(* IEC 61131-3 sources: elnaProjects/kc6/build_BaseProject_ecl/_ (part 4) *)

  errorCMDTimer(In := _commandErrorTimer, PT :=T#90s);

  continueHoldCommandTimer(IN:=(strKr.onStatus = _statusDualInput.STATUS_ON) OR
  (strKr.onStatus = _statusDualInput.STATUS_OFF), PT:=strKr.continueHoldCommand);

  (* ---- алгоритм  для команды ВКЛючить ---- *)
  IF (strKr.onStatus = _statusDualInput.STATUS_ON) and strKr.lastCmdIsOn  then
  	IF strKr.ISVALIDREF_cmdOn AND strKr.ISVALIDREF_cmdOff then
            IF continueHoldCommandTimer.Q THEN
            strKr.cmdOn := false; END_IF;
            END_IF;
  	 errorCMDTimer(In := false);
  	 _commandErrorTimer := false;
  	 cmd_for_Status := 0;
  	 source_for_Status := 0;
  END_IF;

  (* ---- off ---- *)
  IF (strKr.onStatus = _statusDualInput.STATUS_OFF) and  (NOT strKr.lastCmdIsOn) then
  	IF strKr.ISVALIDREF_cmdOn AND strKr.ISVALIDREF_cmdOff then
            IF continueHoldCommandTimer.Q THEN
            strKr.cmdOff := false; END_IF;
            END_IF;
  	 errorCMDTimer(In := false);
  	 _commandErrorTimer := false;
  	 cmd_for_Status := 0;
  	 source_for_Status := 0;
  END_IF;

  (* ---- ошибка исполнения команды ---- *)
  if errorCMDTimer.Q and (cmd_for_Status <> 0) then
  	command_error_for_Status :=  cmd_for_Status;
  	_commandErrorTimer := false;
  	strKr.CmdOn := false;
  	strKr.CmdOff := false;
  	(*lastCmd := 0;*)
  END_IF;

  (* ---- сброс ошибки команды ---- *)
  strKr.CommandFault := command_error_for_Status <> 0;
  _errorReset(IN := command_error_for_Status <> 0, PT := T#5S);
  IF _errorReset.Q THEN
  	cmd_for_Status := 0;
  	source_for_Status := 0;
  	command_error_for_Status := 0;

  END_IF;

  outputsSets(in := (strKr.ISVALIDREF_cmdOn and strKr.cmdOn ) OR (strKr.ISVALIDREF_cmdOff and strKr.cmdOff), PT := T#2S);
  	IF NOT outputsSets.Q THEN
  		strKr.So := inSo._inversed AND inSo.reliability AND strKr.ISVALIDREF_inSo;
  		strKr.Sz := inSz._inversed AND inSz.reliability AND strKr.ISVALIDREF_inSz;
  	END_IF;

  cmdOn := strKr.cmdOn;
  cmdOff:= strKr.cmdOff;

  (* ---- формирование зашифрованного статуса для АРМа ---- *)
  strKr.status := shl(BYTE_TO_DWORD(source_for_Status), 29)
  		OR shl(BYTE_TO_DWORD(cmd_for_Status), 26)
  		OR shl(BYTE_TO_DWORD(command_error_for_Status), 23)
  		OR shl(bool_to_DWORD(strKr.sdvig), 22)
  		OR shl(bool_to_DWORD(strKr.OpcCommandsDisabled), 21)
                      OR shl(bool_to_DWORD(strKr.Dp), 14)
                      OR shl(BOOL_TO_DWORD(strKr.Sz), 13)
  		OR shl(BOOL_TO_DWORD(strKr.So), 12)
  		OR shl(BOOL_TO_DWORD(strKr.ErrorBlock), 11)
  		OR shl(BOOL_TO_DWORD(strKr.ErrorPowerOff), 10)
  		OR shl(BOOL_TO_DWORD(strKr.Manual), 8)
  		OR shl(BOOL_TO_DWORD(strKr.Auto), 7)
  		OR shl(BOOL_TO_DWORD(strKr.Distance), 6)
  		OR shl(BOOL_TO_DWORD(strKr.Local), 5)
  		OR shl(BOOL_TO_DWORD(strKr.Ns), 4)
                  	OR shl(BOOL_TO_DWORD(strKr.Accident ),3)
  		OR BYTE_TO_DWORD(strKr.onStatus);
END_FUNCTION_BLOCK

FUNCTION_BLOCK fb_KranOpenProtectionDual
  VAR_INPUT
    im : struct_Kran;
    dp_konf : struct_AI;
    parametr : struct_DiscretParametr;
  END_VAR
  VAR_IN_OUT
    StrDIp : struct_DiProtection;
  END_VAR
  VAR
    _sunpackerCommand : fb_sunpackerCommand;
    statusDualInput : TYPE_statusDualInput;
    _statusAi : TYPE_StatusAi;
    _ProtectionTags : TYPE_ProtectionTags;
    dP_Konf_izm : LREAL;
    _signalingTp : TOF;
    timer : TON;
    SignalingTrig : R_TRIG;
    SignalingFTrig : F_TRIG;
    SignalingDi : BOOL;
    _signaling : BOOL;
    source : BYTE;
    cmd : BYTE;
    lastCmd : BYTE;
    source_for_Status : BYTE;
    cmd_for_Status : BYTE;
    command_error_for_Status : BYTE;
    resetCmdTimer : TON;
    resetCmdTimerPriznak : BOOL;
    signalinTimer : TON;
    runOnStart_Trig : R_TRIG;
  END_VAR

  IF parametr.Value = 0 THEN
  	dP_Konf_izm:=0.0;
  	timer (in:=(im.onStatus <> statusDualInput.status_on AND
                      ((im.onStatus = statusDualInput.status_off) OR (im.onStatus = statusDualInput.STATUS_TRANSITIONAL))),
                        PT:=StrDIp.delay);
            IF timer.Q THEN
  	    _signaling:=TRUE;
  	ELSE
  	    _signaling:=FALSE;
  	END_IF;

  ELSE
  	timer(in:=FALSE);
  	    IF (im.onStatus <> statusDualInput.status_on) AND
                  ((im.onStatus = statusDualInput.status_off) OR (im.onStatus = statusDualInput.STATUS_TRANSITIONAL)) AND
                   (dP_Konf_izm = 0.0) AND (dp_konf.interval >= _statusAi.Normal) THEN

  		dP_Konf_izm:=dp_konf.value;

  	    ELSIF 	(im.onStatus = statusDualInput.status_on) OR (dp_konf.interval < _statusAi.Normal) THEN
  		dP_Konf_izm:=0.0;
  	    END_IF;

  	    IF	((dP_Konf_izm - dp_konf.value) >= 10.0) AND (dp_konf.interval >= _statusAi.Normal) THEN
  	        _signaling:=TRUE;
  	    ELSE
  	        _signaling:=FALSE;
  	    END_IF;
  END_IF;

  SignalingTrig(CLK := _signaling);
  IF SignalingTrig.Q THEN
  	SignalingDi := TRUE;
  END_IF;
  SignalingFTrig(CLK := _signaling);
  IF SignalingFTrig.Q THEN
  	SignalingDi := FALSE;
  END_IF;

  StrDIp.Tag := StrDIp.inTag;
  StrDIp.RunOnStart := StrDIp.inRunOnStart;

  StrDIp.CanRun := StrDIp.inCanRun;

  StrDIp.OpcCommandsDisabled := StrDIp.inOpcCommandsDisabled;

  (* ---- Если управление с ВУ заблокировано, то передаем команду из алгоритма ---- *)
  IF StrDIp.inOpcCommandsDisabled THEN
  	StrDIp.inCommand := StrDIp.inCommand_Alg;
  ELSE (* иначе передаем команду с АРМа*)
  	StrDIp.inCommand := StrDIp.inCommand_ARM;
  END_IF;

  _sunpackerCommand(command := StrDIp.inCommand);
  	source := _sunpackerCommand.source;
  	cmd := _sunpackerCommand.cmd;

  IF cmd <> 0 AND lastCmd <> cmd AND (((NOT StrDIp.opcCommandsDisabled) AND source > 0) OR source = 0) then
  	CASE BYTE_TO_INT(cmd) OF
  	        (*cmdRun*) 1: 	IF        NOT StrDIp.Remont THEN
  					StrDIp.isEnded := FALSE;
  					StrDIp.hasError 	:= FALSE;
  					StrDIp.isRunning := TRUE;
  					cmd_for_Status := cmd;
  					source_for_Status := source;
  					command_error_for_Status := 0;
  				ELSE
  					StrDIp.isRunning := FALSE;
  					StrDIp.isEnded := FALSE;
  					StrDIp.hasError 	:= FALSE;

  					cmd_for_Status := 0;
  					source_for_Status := source;
  					command_error_for_Status := cmd;
  				END_IF;
                                          StrDIp.inOpcCommandsDisabled:=FALSE;

                  (*cmdReset*) 2: 	StrDIp.isRunning := FALSE;
  				StrDIp.isEnded := FALSE;
  				StrDIp.hasError 	:= FALSE;
  				SignalingDi:= FALSE;
                                          _signaling:=FALSE;
  				StrDIp.Check := FALSE;
  				cmd_for_Status := cmd;
  				source_for_Status := source;
  				command_error_for_Status := 0;
                                          StrDIp.inOpcCommandsDisabled:=FALSE;

  	(*cmd_setRemont*) 4 :	StrDIp.Remont := TRUE;
  				(*StrDIp.isRunning := FALSE;*)

  				cmd_for_Status := cmd;
  				source_for_Status := source;
  				command_error_for_Status := 0;

          (*cmd_resetRemont*) 5 : 	(*IF (im.onStatus<>statusDualInput.STATUS_ON) THEN
  					cmd_for_Status := 0;
  					source_for_Status := 0;
  					command_error_for_Status := cmd;
  				ELSE*)
  					StrDIp.Remont := FALSE;
  					(*StrDIp.isRunning := TRUE;*)

  					cmd_for_Status := cmd;
  					source_for_Status := source;
  					command_error_for_Status := 0;
  				(*END_IF;*)

  	(*cmd_setCheck*) 6 : 	StrDIp.Check := TRUE;

  				cmd_for_Status := cmd;
  				source_for_Status := source;
  				command_error_for_Status := 0;
  	END_CASE;
  	resetCmdTimer(IN := false);
  	resetCmdTimerPriznak := TRUE;
  END_IF;
  lastCmd := cmd;

  resetCmdTimer(IN := resetCmdTimerPriznak);
  IF resetCmdTimer.Q THEN
  	resetCmdTimerPriznak := FALSE;
  	source_for_Status := 0;
  	cmd_for_Status := 0;
  	command_error_for_Status := 0;
  END_IF;

  IF StrDIp.isRunning AND  NOT StrDIp.Remont AND NOT StrDIp.Check THEN
  	StrDIp.Signaling := SignalingDi;
  	StrDIp.SignalingTP := _signalingTp.Q;
  ELSE
  	StrDIp.Signaling := 0;
  	StrDIp.SignalingTP := 0;
  END_IF;

  _signalingTp(in := StrDIp.Signaling, PT := T#1s);

  StrDIp.status :=  SHL(BYTE_TO_DWORD(source_for_Status), 29)
  			OR SHL(BYTE_TO_DWORD(cmd_for_Status), 26)
  			OR SHL(BYTE_TO_DWORD(command_error_for_Status), 23)
  			OR SHL(BOOL_TO_DWORD(StrDIp.OpcCommandsDisabled ), 21)
  			OR SHL(BOOL_TO_DWORD(StrDIp.Signaling), 16)
  			OR SHL(BOOL_TO_DWORD(StrDIp.RunOnStart ), 15)
  			OR SHL(BOOL_TO_DWORD(StrDIp.remont), 6)
  			OR SHL(BOOL_TO_DWORD(StrDIp.Check), 5)
  			OR SHL(BOOL_TO_DWORD(StrDIp.hasError), 4)
  			OR SHL(BOOL_TO_DWORD(StrDIp.SignalingTP), 3)
  			OR SHL(BOOL_TO_DWORD(StrDIp.CanRun), 2)
  			OR SHL(BOOL_TO_DWORD(StrDIp.isEnded), 1)
  			OR BOOL_TO_DWORD(StrDIp.isRunning);
END_FUNCTION_BLOCK

FUNCTION_BLOCK fb_Kran_Init
  VAR_INPUT
    data_Ini : BOOL;
    ISVALIDREF_statOn : BOOL;
    ISVALIDREF_statOff : BOOL;
    ISVALIDREF_cmdOn : BOOL;
    ISVALIDREF_cmdOff : BOOL;
    ISVALIDREF_inSo : BOOL;
    ISVALIDREF_inSz : BOOL;
    ISVALIDREF_inDp : BOOL         := False;
    continueHoldCommand : TIME;
  END_VAR
  VAR_IN_OUT
    str_Kr : struct_Kran;
  END_VAR
  VAR_OUTPUT
    Init : BOOL         := FALSE;
  END_VAR

  (*****            Функциональный блок переинициализации структуры  Kran          *****)

          Init := False;

      IF data_Ini THEN                            (* Параметрам требуется переинициализация. *)
          str_Kr.ISVALIDREF_statOn                := ISVALIDREF_statOn;
          str_Kr.ISVALIDREF_statOff               := ISVALIDREF_statOff;
          str_Kr.ISVALIDREF_cmdOn                 := ISVALIDREF_cmdOn;
          str_Kr.ISVALIDREF_cmdOff                := ISVALIDREF_cmdOff;
          str_Kr.ISVALIDREF_inSo                  := ISVALIDREF_inSo;
          str_Kr.ISVALIDREF_inSz                  := ISVALIDREF_inSz;
          str_Kr.ISVALIDREF_inDp                  := ISVALIDREF_inDp;
          str_Kr.continueHoldCommand              := continueHoldCommand;

          data_Ini:=False;
          Init := TRUE;
     END_IF;
   IF Init THEN
          ISVALIDREF_statOn:= false;
          ISVALIDREF_statOff:= false;
          ISVALIDREF_cmdOn:= false;
          ISVALIDREF_cmdOff:= false;
          ISVALIDREF_inSo:= false;
          ISVALIDREF_inSz:= false;
          ISVALIDREF_inDp:= false;
          continueHoldCommand:= T#0S;
    END_IF;
END_FUNCTION_BLOCK

FUNCTION_BLOCK fb_MvProtectionControlAi
  VAR_INPUT
    sw : struct_SectionSwitch;
  END_VAR
  VAR_IN_OUT
    StrDIp : struct_DiProtection;
  END_VAR
  VAR_INPUT
    ai : struct_AI;
  END_VAR
  VAR
    _sunpackerCommand : fb_sunpackerCommand;
    statusDualInput : TYPE_statusDualInput;
    _statusAi : TYPE_StatusAi;
    _ProtectionTags : TYPE_ProtectionTags;
    _signalingTp : TOF;
    timer : TON;
    SignalingTrig : R_TRIG;
    SignalingFTrig : F_TRIG;
    SignalingDi : BOOL;
    source : BYTE;
    cmd : BYTE;
    lastCmd : BYTE;
    source_for_Status : BYTE;
    cmd_for_Status : BYTE;
    command_error_for_Status : BYTE;
    resetCmdTimer : TON;
    resetCmdTimerPriznak : BOOL;
    signalinTimer : TON;
    runOnStart_Trig : R_TRIG;
  END_VAR

  timer(IN := (sw.onStatus <> statusDualInput.STATUS_ON) AND
              (ai.value < ai.LW) AND (ai.interval >= _statusAi.normal) AND
              StrDIp.isRunning  , PT := StrDIp.delay);

  SignalingTrig(CLK := timer.Q);
  IF SignalingTrig.Q THEN
  	SignalingDi := TRUE;
  END_IF;
  SignalingFTrig(CLK := timer.Q);
  IF SignalingFTrig.Q THEN
  	SignalingDi := FALSE;
  END_IF;

  StrDIp.Tag := StrDIp.inTag;
  StrDIp.RunOnStart := StrDIp.inRunOnStart;

  StrDIp.CanRun := StrDIp.inCanRun;

  StrDIp.OpcCommandsDisabled := StrDIp.inOpcCommandsDisabled;

  (* ---- Если управление с ВУ заблокировано, то передаем команду из алгоритма ---- *)
  IF StrDIp.inOpcCommandsDisabled THEN
  	StrDIp.inCommand := StrDIp.inCommand_Alg;
  ELSE (* иначе передаем команду с АРМа*)
  	StrDIp.inCommand := StrDIp.inCommand_ARM;
  END_IF;

  _sunpackerCommand(command := StrDIp.inCommand);
  	source := _sunpackerCommand.source;
  	cmd := _sunpackerCommand.cmd;

  IF cmd <> 0 AND lastCmd <> cmd AND (((NOT StrDIp.opcCommandsDisabled) AND source > 0) OR source = 0) then
  	CASE BYTE_TO_INT(cmd) OF
  	        (*cmdRun*) 1: 	IF        NOT StrDIp.Remont THEN
  					StrDIp.isEnded := FALSE;
  					StrDIp.hasError 	:= FALSE;
  					StrDIp.isRunning := TRUE;
  					cmd_for_Status := cmd;
  					source_for_Status := source;
  					command_error_for_Status := 0;
  				ELSE
  					StrDIp.isRunning := FALSE;
  					StrDIp.isEnded := FALSE;
  					StrDIp.hasError 	:= FALSE;

  					cmd_for_Status := 0;
  					source_for_Status := source;
  					command_error_for_Status := cmd;
  				END_IF;
                                          StrDIp.inOpcCommandsDisabled:=FALSE;

                  (*cmdReset*) 2: 	StrDIp.isRunning := FALSE;
  				StrDIp.isEnded := FALSE;
  				StrDIp.hasError 	:= FALSE;
  				SignalingDi:= FALSE;
  				StrDIp.Check := FALSE;
  				cmd_for_Status := cmd;
  				source_for_Status := source;
  				command_error_for_Status := 0;
                                          StrDIp.inOpcCommandsDisabled:=FALSE;

  	(*cmd_setRemont*) 4 :	StrDIp.Remont := TRUE;
  				(*StrDIp.isRunning := FALSE;*)

  				cmd_for_Status := cmd;
  				source_for_Status := source;
  				command_error_for_Status := 0;

          (*cmd_resetRemont*) 5 : 	(*IF (sw.onStatus = statusDualInput.STATUS_OFF) THEN
  					cmd_for_Status := 0;
  					source_for_Status := 0;
  					command_error_for_Status := cmd;
  				ELSE*)
  					StrDIp.Remont := FALSE;
  					(*StrDIp.isRunning := TRUE;*)

  					cmd_for_Status := cmd;
  					source_for_Status := source;
  					command_error_for_Status := 0;
  				(*END_IF;*)

  	(*cmd_setCheck*) 6 : 	StrDIp.Check := TRUE;

  				cmd_for_Status := cmd;
  				source_for_Status := source;
  				command_error_for_Status := 0;
  	END_CASE;
  	resetCmdTimer(IN := false);
  	resetCmdTimerPriznak := TRUE;
  END_IF;
  lastCmd := cmd;

  resetCmdTimer(IN := resetCmdTimerPriznak);
  IF resetCmdTimer.Q THEN
  	resetCmdTimerPriznak := FALSE;
  	source_for_Status := 0;
  	cmd_for_Status := 0;
  	command_error_for_Status := 0;
  END_IF;

  IF StrDIp.isRunning AND  NOT StrDIp.Remont AND NOT StrDIp.Check THEN
  	StrDIp.Signaling := SignalingDi;
  	StrDIp.SignalingTP := _signalingTp.Q;
  ELSE
  	StrDIp.Signaling := 0;
  	StrDIp.SignalingTP := 0;
  END_IF;

  _signalingTp(in := StrDIp.Signaling, PT := T#1s);

  StrDIp.status :=  SHL(BYTE_TO_DWORD(source_for_Status), 29)
  			OR SHL(BYTE_TO_DWORD(cmd_for_Status), 26)
  			OR SHL(BYTE_TO_DWORD(command_error_for_Status), 23)
  			OR SHL(BOOL_TO_DWORD(StrDIp.OpcCommandsDisabled ), 21)
  			OR SHL(BOOL_TO_DWORD(StrDIp.Signaling), 16)
  			OR SHL(BOOL_TO_DWORD(StrDIp.RunOnStart ), 15)
  			OR SHL(BOOL_TO_DWORD(StrDIp.remont), 6)
  			OR SHL(BOOL_TO_DWORD(StrDIp.Check), 5)
  			OR SHL(BOOL_TO_DWORD(StrDIp.hasError), 4)
  			OR SHL(BOOL_TO_DWORD(StrDIp.SignalingTP), 3)
  			OR SHL(BOOL_TO_DWORD(StrDIp.CanRun), 2)
  			OR SHL(BOOL_TO_DWORD(StrDIp.isEnded), 1)
  			OR BOOL_TO_DWORD(StrDIp.isRunning);
END_FUNCTION_BLOCK

FUNCTION_BLOCK fb_OilPump_Init
  VAR_INPUT
    data_Ini : BOOL;
    ISVALIDREF_statOn : BOOL;
    ISVALIDREF_statOff : BOOL;
    ISVALIDREF_cmdOn : BOOL;
    ISVALIDREF_cmdOff : BOOL;
    ISVALIDREF_inBreakCmdOn : BOOL;
    ISVALIDREF_inBreakCmdOff : BOOL;
  END_VAR
  VAR_IN_OUT
    str_Op : struct_OilPump;
  END_VAR
  VAR_OUTPUT
    Init : BOOL         := FALSE;
  END_VAR

  (*****            Функциональный блок переинициализации структуры  НУ          *****)

   Init := FALSE;

      IF data_Ini THEN                            (* Параметрам требуется переинициализация. *)
          str_Op.ISVALIDREF_statOn                := ISVALIDREF_statOn;
          str_Op.ISVALIDREF_statOff               := ISVALIDREF_statOff;
          str_Op.ISVALIDREF_cmdOn                 := ISVALIDREF_cmdOn;
          str_Op.ISVALIDREF_cmdOff                := ISVALIDREF_cmdOff;
          str_Op.ISVALIDREF_inBreakCmdOn          := ISVALIDREF_inBreakCmdOn;
          str_Op.ISVALIDREF_inBreakCmdOff         := ISVALIDREF_inBreakCmdOff;
          data_Ini:=FALSE;
          Init := TRUE;
      END_IF;

          ISVALIDREF_statOn:= FALSE;
          ISVALIDREF_statOff:= FALSE;
          ISVALIDREF_cmdOn:= FALSE;
          ISVALIDREF_cmdOff:= FALSE;
          ISVALIDREF_inBreakCmdOn:= FALSE;
          ISVALIDREF_inBreakCmdOff:= FALSE;
END_FUNCTION_BLOCK

FUNCTION_BLOCK fb_ProtectionsManager
  VAR
    cmd : BYTE;
  END_VAR
  VAR_IN_OUT
    str_PM : struct_ProtectionsManager;
  END_VAR
  VAR
    lastCmd : BYTE;
    autoRunPriznak : BOOL;
    onInit : BOOL;
  END_VAR
  VAR_EXTERNAL
    protections : ProtectionsConfig;
  END_VAR
  VAR
    timerUnBlock : TON;
    timerAutoRun : TON;
    UnBlockPriznak : BOOL;
  END_VAR

  IF NOT onInit THEN

      autoRunProtections(protections);
  onInit:=TRUE;
  END_IF;

  str_PM.protectionInRemont:=anyProtectioninRemont(protections);

  cmd := str_PM.inCommand;

  IF cmd <> 0 AND lastCmd <> cmd then
                UnBlockPriznak:=TRUE;
  	CASE BYTE_TO_INT(cmd) OF

  		(*RestartAllSignaling*) 1: 	ResetAllSignaling(protections);
  				          autoRunPriznak:=TRUE;

  	        (*RestartAllProtections*) 2: 	ResetAllProtections(protections);
                                                    autoRunPriznak:=TRUE;

                        (*CheckProtections*)  3: 	RunAllProtections(protections);

  	         (*ResetAllProtections*)  4: 	ResetAllProtections(protections);

  	END_CASE;

  END_IF;
  lastCmd := cmd;
  timerUnBlock(IN:=UnBlockPriznak, PT:=T#1S);
  timerAutoRun(IN:=autoRunPriznak, PT:=T#500MS);

  IF timerAutoRun.Q THEN autoRunProtections(protections);
  END_IF;

  IF timerUnBlock.Q THEN
  lastCmd:= 0;
  str_PM.inCommand:=0;
  autoRunPriznak:=FALSE;
  UnBlockPriznak:=FALSE;
  END_IF;
END_FUNCTION_BLOCK

FUNCTION_BLOCK fb_SectionSwitch
  VAR_INPUT
    statOn : BOOL;
    statOff : BOOL;
    statOn_reliability : BOOL;
    statOff_reliability : BOOL;
  END_VAR
  VAR_IN_OUT
    StrSw : struct_SectionSwitch;
  END_VAR
  VAR_INPUT
    basketRolledIn : TYPE_ReliableBit;
    basketRolledOut : TYPE_ReliableBit;
    basketTest : TYPE_ReliableBit;
    inNs : TYPE_ReliableBit;
    inoffKNA : TYPE_ReliableBit;
    inAccident : TYPE_ReliableBit;
    inLocal : TYPE_ReliableBit;
    inDistance : TYPE_ReliableBit;
    inBreakCmdOn : TYPE_ReliableBit;
    inBreakCmdOff : TYPE_ReliableBit;
  END_VAR
  VAR
    onInit : BOOL         := FALSE;
    _statOn : BOOL;
    _statOff : BOOL;
    lastOnStatus : BYTE;
    cmd : BYTE;
    source : BYTE;
    lastCmd : BYTE;
    source_for_Status : BYTE;
    cmd_for_Status : BYTE;
    command_error_for_Status : BYTE;
    _basketRolledIn : TYPE_ReliableBit;
    _basketRolledOut : TYPE_ReliableBit;
    _basketTest : TYPE_ReliableBit;
    _sunpackerCommand : fb_sunpackerCommand;
    _statusDualInput : TYPE_statusDualInput;
    _statusBasket : TYPE_basketStats;
    _commandDualInput : TYPE_commandDualInput;
    _commandErrorTimer : BOOL;
    resetErrorTimer : BOOL;
    _changWithoutCommand : BOOL;
    errorCMDTimer : TON;
    _errorReset : TON;
    outputsSets : TOF;
  END_VAR
  VAR_IN_OUT
    cmdOn : BOOL;
    cmdOff : BOOL;
  END_VAR

  IF NOT onInit THEN
  IF StrSw.ISVALIDREF_cmdOn XOR StrSw.ISVALIDREF_cmdOff THEN
  	IF 	StrSw.ISVALIDREF_cmdOn THEN
  		lastCmd:= 2; (*baseCmdOff*)
  	ELSE
  		lastCmd:= 1; (*baseCmdOn*)
  	END_IF;
  END_IF;
  onInit:=TRUE;
  END_IF;

  (* ---- Формирование состояния тележки ---- *)

  IF (NOT StrSw.ISVALIDREF_basketRolledIn) AND (NOT StrSw.ISVALIDREF_basketRolledOut) THEN
            StrSw.basketStatus:=_statusBasket.BASKET_NOTDEFINED;
  ELSE
  		IF StrSw.ISVALIDREF_basketTest THEN
  		_basketTest:=basketTest;
  	ELSE
  		_basketTest.reliability:=TRUE;
  		_basketTest.value :=FALSE;
  	END_IF;

  	IF StrSw.ISVALIDREF_basketRolledIn THEN
  		_basketRolledIn:=basketRolledIn;
  	ELSE
  		_basketRolledIn:=basketRolledOut;
  		IF StrSw.ISVALIDREF_basketTest THEN
  		_basketRolledIn.value:=NOT (_basketRolledIn.value OR _basketTest.value);
  		ELSE
  		_basketRolledIn.value:= NOT _basketRolledIn.value;
  		END_IF;

  	END_IF;

  	IF StrSw.ISVALIDREF_basketRolledOut THEN
  		_basketRolledOut:=basketRolledOut;
  	ELSE
  		_basketRolledOut:=basketRolledIn;
  		IF StrSw.ISVALIDREF_basketTest THEN
  		_basketRolledOut.value:= NOT (_basketRolledOut.value OR _basketTest.value );
  		ELSE
  			_basketRolledOut.value := NOT _basketRolledout.value;
  		END_IF;

  	END_IF;

  IF _basketRolledIn.reliability AND _basketRolledOut.reliability AND _basketTest.reliability THEN
  		IF (BOOL_TO_INT(_basketRolledIn.value)+BOOL_TO_INT(_basketRolledOut.value)+BOOL_TO_INT(_basketTest.value))=1 THEN
  			IF _basketRolledIn.value THEN
  				StrSw.basketStatus:=_statusBasket.BASKET_ROLLEDIN;
  			ELSIF _basketRolledOut.value THEN
  				StrSw.basketStatus:=_statusBasket.BASKET_ROLLEDOUT;
  			ELSIF _basketTest.value THEN
  				StrSw.basketStatus:=_statusBasket.BASKET_TEST;
  			END_IF;
  		ELSE
  			StrSw.basketStatus:=_statusBasket.BASKET_ERROR;
  		END_IF;
  	ELSE
  		StrSw.basketStatus:=_statusBasket.BASKET_NOTDEFINED;
  	END_IF;
  END_IF;

  (* ---- Если управление с ВУ заблокировано, то в ИМ передаем команду из алгоритма ---- *)
  IF StrSw.inOpcCommandsDisabled THEN
  	StrSw.inCommand := StrSw.inCommand_Alg;
  ELSE (* иначе передаем команду с АРМа*)
  	StrSw.inCommand := StrSw.inCommand_ARM;
  END_IF;

  (* ---- Формирование состояния механизма ---- *)

  IF (StrSw.ISVALIDREF_statOn) OR (StrSw.ISVALIDREF_statOff) THEN
  	IF (StrSw.ISVALIDREF_statOn) AND (StrSw.ISVALIDREF_statOff) THEN
  	StrSw.reliability:= statOn_reliability AND statOff_reliability;
  		_statOn  := statOn;
  		_statOff := statOff;
  	ELSIF (StrSw.ISVALIDREF_statOn) THEN
                       StrSw.reliability:= statOn_reliability;
  		_statOn  := statOn;
  		_statOff := NOT statOn;
  	ELSIF (StrSw.ISVALIDREF_statOff) THEN
  		 StrSw.reliability:= statOff_reliability;
  		_statOn  := NOT statOff;
  		_statOff :=statOff;
  	END_IF;

  	IF StrSw.reliability THEN
  		IF _statOn AND NOT _statOff 		THEN 	StrSw.onStatus := _statusDualInput.STATUS_ON;
  		ELSIF _statOff AND NOT _statOn 	THEN 	StrSw.onStatus := _statusDualInput.Status_OFF;
  		ELSIF NOT _statOn AND NOT _statOff 	THEN 	StrSw.onStatus := _statusDualInput.STATUS_TRANSITIONAL;
  		ELSE					StrSw.onStatus := _statusDualInput.STATUS_ERROR;
                      END_IF;

  	ELSE
  		StrSw.onStatus := _statusDualInput.STATUS_NOTDEFINED;

  	END_IF;
  ELSE
  	CASE BYTE_TO_INT(lastCmd) OF
  		(*baseCmdOn*) 1: StrSw.onStatus  := _statusDualInput.STATUS_ON;
  		(*baseCmdOff*) 2: StrSw.onStatus  := _statusDualInput.STATUS_OFF;

  	ELSE
  		 StrSw.onStatus := _statusDualInput.STATUS_NOTDEFINED;

  	END_CASE;
  END_IF;

  StrSw.Accident := inAccident.value AND inAccident.reliability;
  StrSw.Ns := inNs.value AND inNs.reliability;
  StrSw.Local := inLocal.value AND inLocal.reliability;
  StrSw.Distance := inDistance.value AND inDistance.reliability;
  StrSw.OpcCommandsDisabled := StrSw.inOpcCommandsDisabled;
  StrSw.offKNA := inoffKNA.value AND inoffKNA.reliability;
  (* ---- Формирование признака сдвига ---- *)
  StrSw.sdvig  := FALSE;
  IF (StrSw.ISVALIDREF_cmdOn OR StrSw.ISVALIDREF_cmdOff) AND NOT StrSw.Local THEN
  	IF cmd = 0 THEN
  		IF (lastOnStatus <> StrSw.onStatus AND
  		(StrSw.onStatus <> _statusDualInput.STATUS_NOTDEFINED AND StrSw.onStatus <> _statusDualInput.STATUS_ERROR) AND
  		(lastOnStatus <> _statusDualInput.STATUS_NOTDEFINED AND lastOnStatus <> _statusDualInput.STATUS_ERROR)) THEN
  			StrSw.sdvig   := TRUE;
  		END_IF;
  	END_IF;
  END_IF;
  lastOnStatus := StrSw.onStatus;

  (* ---- Распаковка команды ---- *)
  _sunpackerCommand(command := StrSw.inCommand);
  	cmd := _sunpackerCommand.cmd;
  	source := _sunpackerCommand.source;

  (* ---- Обработка команды ---- *)
  IF cmd <> 0 AND lastCmd <> cmd and (((NOT StrSw.opcCommandsDisabled) AND source > 0) OR source = 0) then
  	CASE BYTE_TO_INT(cmd) OF
  	(*cmd_open*) 1 :
  			IF  StrSw.ISVALIDREF_cmdOn THEN StrSw.CmdOn := TRUE;
  				IF StrSw.ISVALIDREF_cmdOff THEN StrSw.CmdOff := FALSE; END_IF;
  			ELSIF  StrSw.ISVALIDREF_cmdOff THEN StrSw.CmdOff := FALSE;  END_IF;
  			errorCMDTimer(IN := false);
  			_commandErrorTimer := true;
  			StrSw.lastCmdIsOn := true;
  	(*cmd_close*) 2 :
  			IF StrSw.ISVALIDREF_cmdOff THEN StrSw.CmdOff := TRUE;
  				IF StrSw.ISVALIDREF_cmdOn THEN StrSw.CmdOn := FALSE; END_IF;
  			ELSIF StrSw.ISVALIDREF_cmdOn THEN StrSw.CmdOn := FALSE; END_IF;
  			errorCMDTimer(IN := false);
  			_commandErrorTimer := true;
  			StrSw.lastCmdIsOn := false;
  	(*cmd_reset*) 3 :    IF StrSw.ISVALIDREF_statOn OR StrSw.ISVALIDREF_statOff THEN
  			StrSw.CmdOn := FALSE;
  			StrSw.CmdOff := FALSE;
                                lastCmd := 0;
  			_commandErrorTimer := false;
  			StrSw.lastCmdIsOn := false;
                                 END_IF;
  	END_CASE;
  	source_for_Status := source;
  	cmd_for_Status := cmd;
  	command_error_for_Status := 0;
  END_IF;
  lastCmd := cmd;

  errorCMDTimer(In := _commandErrorTimer, PT :=T#10s);

  (* ---- алгоритм  для команды ВКЛючить ---- *)
  IF (StrSw.onStatus = _statusDualInput.STATUS_ON) and (StrSw.lastCmdIsOn) then
  	IF StrSw.ISVALIDREF_cmdOn AND StrSw.ISVALIDREF_cmdOff then  StrSw.cmdOn := false; END_IF;

  	 errorCMDTimer(In := false);
  	 _commandErrorTimer := false;
  	 cmd_for_Status := 0;
  	 source_for_Status := 0;
  END_IF;

  (* ---- off ---- *)
  IF (StrSw.onStatus = _statusDualInput.STATUS_OFF) and (NOT StrSw.lastCmdIsOn) then
  	IF StrSw.ISVALIDREF_cmdOn AND StrSw.ISVALIDREF_cmdOff then  StrSw.cmdOff := false; END_IF;

  	 errorCMDTimer(In := false);
  	 _commandErrorTimer := false;
  	 cmd_for_Status := 0;
  	 source_for_Status := 0;
  END_IF;

  (* ---- ошибка исполнения команды ---- *)
  if errorCMDTimer.Q and (cmd_for_Status <> 0) then
  	command_error_for_Status :=  cmd_for_Status;
  	_commandErrorTimer := false;
  	StrSw.CmdOn := false;
  	StrSw.CmdOff := false;
  	lastCmd := 0;
  end_if;

  (* ---- сброс ошибки команды ---- *)
  StrSw.CommandFault := command_error_for_Status <> 0;
  _errorReset(IN := command_error_for_Status <> 0, PT := T#5S);
  IF _errorReset.Q THEN
  	cmd_for_Status := 0;
  	source_for_Status := 0;
  	command_error_for_Status := 0;
  END_IF;

  outputsSets(in := (StrSw.ISVALIDREF_cmdOn and StrSw.cmdOn ) OR (StrSw.ISVALIDREF_cmdOff and StrSw.cmdOff), PT := T#2S);
  	IF NOT outputsSets.Q THEN
  		StrSw.BreakCmdOn := inBreakCmdOn._inversed AND inBreakCmdOn.reliability AND StrSw.ISVALIDREF_inBreakCmdOn;
  		StrSw.BreakCmdOff := inBreakCmdOff._inversed AND inBreakCmdOff.reliability AND StrSw.ISVALIDREF_inBreakCmdOff;
  	END_IF;

  cmdOn := StrSw.cmdOn;
  cmdOff:= StrSw.cmdOff;

  (* ---- формирование зашифрованного статуса для АРМа ---- *)
  StrSw.status := shl(BYTE_TO_DWORD(source_for_Status), 29)
  		OR shl(BYTE_TO_DWORD(cmd_for_Status), 26)
  		OR shl(BYTE_TO_DWORD(command_error_for_Status), 23)
  		OR shl(bool_to_DWORD(StrSw.sdvig), 22)
  		OR shl(bool_to_DWORD(StrSw.OpcCommandsDisabled), 21)
                      OR shl(BOOL_TO_DWORD(StrSw.offKNA), 17)
                      OR shl(bool_to_DWORD(StrSw.lastCmdIsOn), 14)
                      OR shl(BOOL_TO_DWORD(StrSw.BreakCmdOff), 13)
  		OR shl(BOOL_TO_DWORD(StrSw.BreakCmdOn), 12)
                      OR shl(BYTE_TO_DWORD(StrSw.basketStatus), 8)
  		OR shl(BOOL_TO_DWORD(StrSw.Distance), 6)
  		OR shl(BOOL_TO_DWORD(StrSw.Local), 5)
  		OR shl(BOOL_TO_DWORD(StrSw.Ns), 4)
                  	OR shl(BOOL_TO_DWORD(StrSw.Accident ),3)
  		OR BYTE_TO_DWORD(StrSw.onStatus);
END_FUNCTION_BLOCK

FUNCTION_BLOCK fb_SectionSwitch_Init
  VAR_INPUT
    data_Ini : BOOL;
    ISVALIDREF_statOn : BOOL;
    ISVALIDREF_statOff : BOOL;
    ISVALIDREF_cmdOn : BOOL;
    ISVALIDREF_cmdOff : BOOL;
    ISVALIDREF_inBreakCmdOn : BOOL;
    ISVALIDREF_inBreakCmdOff : BOOL;
    ISVALIDREF_basketRolledIn : BOOL;
    ISVALIDREF_basketRolledOut : BOOL;
    ISVALIDREF_basketTest : BOOL;
  END_VAR
  VAR_IN_OUT
    str_Sw : struct_SectionSwitch;
  END_VAR
  VAR_OUTPUT
    Init : BOOL         := FALSE;
  END_VAR

  (*****            Функциональный блок переинициализации структуры  МВ          *****)

   Init := FALSE;

      IF data_Ini THEN                            (* Параметрам требуется переинициализация. *)
          str_Sw.ISVALIDREF_statOn                := ISVALIDREF_statOn;
          str_Sw.ISVALIDREF_statOff               := ISVALIDREF_statOff;
          str_Sw.ISVALIDREF_cmdOn                 := ISVALIDREF_cmdOn;
          str_Sw.ISVALIDREF_cmdOff                := ISVALIDREF_cmdOff;
          str_Sw.ISVALIDREF_inBreakCmdOn          := ISVALIDREF_inBreakCmdOn;
          str_Sw.ISVALIDREF_inBreakCmdOff         := ISVALIDREF_inBreakCmdOff;
          str_Sw.ISVALIDREF_basketRolledIn        := ISVALIDREF_basketRolledIn;
          str_Sw.ISVALIDREF_basketRolledOut       := ISVALIDREF_basketRolledOut;
          str_Sw.ISVALIDREF_basketTest            := ISVALIDREF_basketTest;
          data_Ini:=FALSE;
          Init := TRUE;
      END_IF;
  IF Init THEN
          ISVALIDREF_statOn:= FALSE;
          ISVALIDREF_statOff:= FALSE;
          ISVALIDREF_cmdOn:= FALSE;
          ISVALIDREF_cmdOff:= FALSE;
          ISVALIDREF_inBreakCmdOn:= FALSE;
          ISVALIDREF_inBreakCmdOff:= FALSE;
          ISVALIDREF_basketRolledIn:= FALSE;
          ISVALIDREF_basketRolledOut:= FALSE;
          ISVALIDREF_basketTest:= FALSE;
  END_IF;
END_FUNCTION_BLOCK

FUNCTION_BLOCK fb_Switch
  VAR_INPUT
    statOn : BOOL;
    statOff : BOOL;
    statOn_reliability : BOOL;
    statOff_reliability : BOOL;
  END_VAR
  VAR_IN_OUT
    StrSw : struct_Switch;
  END_VAR
  VAR_INPUT
    inNs : TYPE_ReliableBit;
    inAccident : TYPE_ReliableBit;
    inAuto : TYPE_ReliableBit;
    inManual : TYPE_ReliableBit;
    inLocal : TYPE_ReliableBit;
    inDistance : TYPE_ReliableBit;
    inErrorPowerOff : TYPE_ReliableBit;
    inErrorBlock : TYPE_ReliableBit;
    inBreakCmdOn : TYPE_ReliableBit;
    inBreakCmdOff : TYPE_ReliableBit;
  END_VAR
  VAR
    onInit : BOOL         := FALSE;
    _reliability : BOOL;
    _statOn : BOOL;
    _statOff : BOOL;
    lastOnStatus : BYTE;
    cmd : BYTE;
    source : BYTE;
    lastCmd : BYTE;
    source_for_Status : BYTE;
    cmd_for_Status : BYTE;
    command_error_for_Status : BYTE;
    _sunpackerCommand : fb_sunpackerCommand;
    _statusDualInput : TYPE_statusDualInput;
    _commandDualInput : TYPE_commandDualInput;
    _commandErrorTimer : BOOL;
    resetErrorTimer : BOOL;
    _changWithoutCommand : BOOL;
    errorCMDTimer : TON;
    _errorReset : TON;
    outputsSets : TOF;
  END_VAR
  VAR_IN_OUT
    cmdOn : BOOL;
    cmdOff : BOOL;
  END_VAR

  IF NOT onInit THEN
  IF StrSw.ISVALIDREF_cmdOn XOR StrSw.ISVALIDREF_cmdOff THEN
  	IF 	StrSw.ISVALIDREF_cmdOn THEN
  		lastCmd:= 2; (*baseCmdOff*)
  	ELSE
  		lastCmd:= 1; (*baseCmdOn*)
  	END_IF;
  END_IF;
  onInit:=TRUE;
  END_IF;

  (* ---- Если управление с ВУ заблокировано, то в ИМ передаем команду из алгоритма ---- *)
  IF StrSw.inOpcCommandsDisabled THEN
  	StrSw.inCommand := StrSw.inCommand_Alg;
  ELSE (* иначе передаем команду с АРМа*)
  	StrSw.inCommand := StrSw.inCommand_ARM;
  END_IF;

  (* ---- Формирование состояния механизма ---- *)

  IF (StrSw.ISVALIDREF_statOn) OR (StrSw.ISVALIDREF_statOff) THEN
  	IF (StrSw.ISVALIDREF_statOn) AND (StrSw.ISVALIDREF_statOff) THEN
  	_reliability:= statOn_reliability AND statOff_reliability;
  		_statOn  := statOn;
  		_statOff := statOff;
  	ELSIF (StrSw.ISVALIDREF_statOn) THEN
                       _reliability:= statOn_reliability;
  		_statOn  := statOn;
  		_statOff := NOT statOn;
  	ELSIF (StrSw.ISVALIDREF_statOff) THEN
  		 _reliability:= statOff_reliability;
  		_statOn  := NOT statOff;
  		_statOff :=statOff;
  	END_IF;

  	IF _reliability THEN
  		IF _statOn AND NOT _statOff 		THEN 	StrSw.onStatus := _statusDualInput.STATUS_ON;
  		ELSIF _statOff AND NOT _statOn 	THEN 	StrSw.onStatus := _statusDualInput.Status_OFF;
  		ELSIF NOT _statOn AND NOT _statOff 	THEN 	StrSw.onStatus := _statusDualInput.STATUS_TRANSITIONAL;
  		ELSE					StrSw.onStatus := _statusDualInput.STATUS_ERROR;
                      END_IF;

  	ELSE
  		StrSw.onStatus := _statusDualInput.STATUS_NOTDEFINED;

  	END_IF;
  ELSE
  	CASE BYTE_TO_INT(lastCmd) OF
  		(*baseCmdOn*) 1: StrSw.onStatus  := _statusDualInput.STATUS_ON;
  		(*baseCmdOff*) 2: StrSw.onStatus  := _statusDualInput.STATUS_OFF;

  	ELSE
  		 StrSw.onStatus := _statusDualInput.STATUS_NOTDEFINED;

  	END_CASE;
  END_IF;

  StrSw.Accident := inAccident.value AND inAccident.reliability;
  StrSw.Ns := inNs.value AND inNs.reliability;
  StrSw.Auto := inAuto.value AND inAuto.reliability;
  StrSw.Manual := inManual.value AND inManual.reliability;
  StrSw.Local := inLocal.value AND inLocal.reliability;
  StrSw.Distance := inDistance.value AND inDistance.reliability;
  StrSw.ErrorPowerOff := inErrorPowerOff.value AND inErrorPowerOff.reliability;
  StrSw.ErrorBlock := inErrorBlock.value AND inErrorBlock.reliability;
  StrSw.OpcCommandsDisabled := StrSw.inOpcCommandsDisabled;

  (* ---- Формирование признака сдвига ---- *)
  StrSw.sdvig  := FALSE;
  IF (StrSw.ISVALIDREF_cmdOn OR StrSw.ISVALIDREF_cmdOff) AND NOT StrSw.Local THEN
  	IF cmd = 0 THEN
  		IF (lastOnStatus <> StrSw.onStatus AND
  		(StrSw.onStatus <> _statusDualInput.STATUS_NOTDEFINED AND StrSw.onStatus <> _statusDualInput.STATUS_ERROR) AND
  		(lastOnStatus <> _statusDualInput.STATUS_NOTDEFINED AND lastOnStatus <> _statusDualInput.STATUS_ERROR)) THEN
  			StrSw.sdvig   := TRUE;
  		END_IF;
  	END_IF;
  END_IF;
  lastOnStatus := StrSw.onStatus;

  (* ---- Распаковка команды ---- *)
  _sunpackerCommand(command := StrSw.inCommand);
  	cmd := _sunpackerCommand.cmd;
  	source := _sunpackerCommand.source;

  (* ---- Обработка команды ---- *)
  IF cmd <> 0 AND lastCmd <> cmd and (((NOT StrSw.opcCommandsDisabled) AND source > 0) OR source = 0) then
  	CASE BYTE_TO_INT(cmd) OF
  	(*cmd_open*) 1 :
  			IF  StrSw.ISVALIDREF_cmdOn THEN StrSw.CmdOn := TRUE;
  				IF StrSw.ISVALIDREF_cmdOff THEN StrSw.CmdOff := FALSE; END_IF;
  			ELSIF  StrSw.ISVALIDREF_cmdOff THEN StrSw.CmdOff := FALSE;  END_IF;
  			errorCMDTimer(IN := false);
  			_commandErrorTimer := true;
  			StrSw.lastCmdIsOn := true;
  	(*cmd_close*) 2 :
  			IF StrSw.ISVALIDREF_cmdOff THEN StrSw.CmdOff := TRUE;
  				IF StrSw.ISVALIDREF_cmdOn THEN StrSw.CmdOn := FALSE; END_IF;
  			ELSIF StrSw.ISVALIDREF_cmdOn THEN StrSw.CmdOn := FALSE; END_IF;
  			errorCMDTimer(IN := false);

  			_commandErrorTimer := true;
  			StrSw.lastCmdIsOn := false;
  	(*cmd_reset*) 3 :    IF StrSw.ISVALIDREF_statOn OR StrSw.ISVALIDREF_statOff THEN
  			StrSw.CmdOn := FALSE;
  			StrSw.CmdOff := FALSE;
                                lastCmd :=0;
  			_commandErrorTimer := false;
  			StrSw.lastCmdIsOn := false;
                                 END_IF;
  	END_CASE;
  	source_for_Status := source;
  	cmd_for_Status := cmd;
  	command_error_for_Status := 0;
  END_IF;

  lastCmd := cmd;
  errorCMDTimer(In := _commandErrorTimer, PT :=T#10s);

  (* ---- алгоритм  для команды ВКЛючить ---- *)
  IF (StrSw.onStatus = _statusDualInput.STATUS_ON) and StrSw.lastCmdIsOn then
  	IF StrSw.ISVALIDREF_cmdOn AND StrSw.ISVALIDREF_cmdOff then  StrSw.cmdOn := false; END_IF;

  	 errorCMDTimer(In := false);
  	 _commandErrorTimer := false;
  	 cmd_for_Status := 0;
  	 source_for_Status := 0;
  END_IF;

  (* ---- off ---- *)
  IF (StrSw.onStatus = _statusDualInput.STATUS_OFF) and (NOT StrSw.lastCmdIsOn) then
  	IF StrSw.ISVALIDREF_cmdOn AND StrSw.ISVALIDREF_cmdOff then  StrSw.cmdOff := false; END_IF;

  	 errorCMDTimer(In := false);
  	 _commandErrorTimer := false;
  	 cmd_for_Status := 0;
  	 source_for_Status := 0;
  END_IF;

  (* ---- ошибка исполнения команды ---- *)
  if errorCMDTimer.Q and (cmd_for_Status <> 0) then
  	command_error_for_Status :=  cmd_for_Status;
  	_commandErrorTimer := false;
  	StrSw.CmdOn := false;
  	StrSw.CmdOff := false;
  	lastCmd := 0;
  end_if;

  (* ---- сброс ошибки команды ---- *)
  StrSw.CommandFault := command_error_for_Status <> 0;
  _errorReset(IN := command_error_for_Status <> 0, PT := T#5S);
  IF _errorReset.Q THEN
  	cmd_for_Status := 0;
  	source_for_Status := 0;
  	command_error_for_Status := 0;
  END_IF;

  outputsSets(in := (StrSw.ISVALIDREF_cmdOn and StrSw.cmdOn ) OR (StrSw.ISVALIDREF_cmdOff and StrSw.cmdOff), PT := T#2S);
  	IF NOT outputsSets.Q THEN
  		StrSw.BreakCmdOn := inBreakCmdOn._inversed AND inBreakCmdOn.reliability AND StrSw.ISVALIDREF_inBreakCmdOn;
  		StrSw.BreakCmdOff := inBreakCmdOff._inversed AND inBreakCmdOff.reliability AND StrSw.ISVALIDREF_inBreakCmdOff;
  	END_IF;

  cmdOn := StrSw.cmdOn;
  cmdOff:= StrSw.cmdOff;

  (* ---- формирование зашифрованного статуса для АРМа ---- *)
  StrSw.status := shl(BYTE_TO_DWORD(source_for_Status), 29)
  		OR shl(BYTE_TO_DWORD(cmd_for_Status), 26)
  		OR shl(BYTE_TO_DWORD(command_error_for_Status), 23)
  		OR shl(bool_to_DWORD(StrSw.sdvig), 22)
  		OR shl(bool_to_DWORD(StrSw.OpcCommandsDisabled), 21)
                      OR shl(bool_to_DWORD(StrSw.lastCmdIsOn), 14)
                      OR shl(BOOL_TO_DWORD(StrSw.BreakCmdOff), 13)
  		OR shl(BOOL_TO_DWORD(StrSw.BreakCmdOn), 12)
  		OR shl(BOOL_TO_DWORD(StrSw.ErrorBlock), 11)
  		OR shl(BOOL_TO_DWORD(StrSw.ErrorPowerOff), 10)
  		OR shl(BOOL_TO_DWORD(StrSw.Manual), 8)
  		OR shl(BOOL_TO_DWORD(StrSw.Auto), 7)
  		OR shl(BOOL_TO_DWORD(StrSw.Distance), 6)
  		OR shl(BOOL_TO_DWORD(StrSw.Local), 5)
  		OR shl(BOOL_TO_DWORD(StrSw.Ns), 4)
                  	OR shl(BOOL_TO_DWORD(StrSw.Accident ),3)
  		OR BYTE_TO_DWORD(StrSw.onStatus);
END_FUNCTION_BLOCK

FUNCTION_BLOCK fb_Switch_Init
  VAR_INPUT
    data_Ini : BOOL;
    ISVALIDREF_statOn : BOOL;
    ISVALIDREF_statOff : BOOL;
    ISVALIDREF_cmdOn : BOOL;
    ISVALIDREF_cmdOff : BOOL;
    ISVALIDREF_inBreakCmdOn : BOOL;
    ISVALIDREF_inBreakCmdOff : BOOL;
  END_VAR
  VAR_IN_OUT
    str_Sw : struct_Switch;
  END_VAR
  VAR_OUTPUT
    Init : BOOL         := FALSE;
  END_VAR

  (*****            Функциональный блок переинициализации структуры  Switch          *****)

   Init := FALSE;

      IF data_Ini THEN                            (* Параметрам требуется переинициализация. *)
          str_Sw.ISVALIDREF_statOn                := ISVALIDREF_statOn;
          str_Sw.ISVALIDREF_statOff               := ISVALIDREF_statOff;
          str_Sw.ISVALIDREF_cmdOn                 := ISVALIDREF_cmdOn;
          str_Sw.ISVALIDREF_cmdOff                := ISVALIDREF_cmdOff;
          str_Sw.ISVALIDREF_inBreakCmdOn          := ISVALIDREF_inBreakCmdOn;
          str_Sw.ISVALIDREF_inBreakCmdOff         := ISVALIDREF_inBreakCmdOff;
          data_Ini:=FALSE;
          Init := TRUE;
      END_IF;
  IF Init THEN
          ISVALIDREF_statOn:= FALSE;
          ISVALIDREF_statOff:= FALSE;
          ISVALIDREF_cmdOn:= FALSE;
          ISVALIDREF_cmdOff:= FALSE;
          ISVALIDREF_inBreakCmdOn:= FALSE;
          ISVALIDREF_inBreakCmdOff:= FALSE;
  END_IF;
END_FUNCTION_BLOCK

FUNCTION_BLOCK fb_meandr
  VAR
    _output : BOOL;
  END_VAR
  VAR_INPUT
    period : TIME         := T#300MS;
  END_VAR
  VAR
    timer : TON;
    FALSE_val : BOOL         := FALSE;
    TRUE_val : BOOL         := TRUE;
  END_VAR
  VAR_IN_OUT
    output : BOOL;
  END_VAR

  timer(in:=NOT FALSE_val,PT:=period);

  IF timer.Q THEN
      _output:=_output XOR TRUE_val;
      timer(in:=FALSE);
  END_IF;

  output:=_output;
END_FUNCTION_BLOCK

FUNCTION_BLOCK fb_puskOilSystemAlg
  VAR_IN_OUT
    StrAlg : struct_Alg;
  END_VAR
  VAR
    pnsOn : struct_PhaseAlgoritm;
    LowOil : struct_PhaseAlgoritm;
    BreakPuskTimer_Poil : struct_PhaseAlgoritm;
    Poil_DefenseActive : struct_PhaseAlgoritm;
    autoNuOn : struct_PhaseAlgoritm;
    nuOn : struct_PhaseAlgoritm;
    nu1On : struct_PhaseAlgoritm;
    nu2On : struct_PhaseAlgoritm;
    di_dPmg : struct_PhaseAlgoritm;
    dP_oilGas100 : struct_PhaseAlgoritm;
    runProtect_dP : struct_PhaseAlgoritm;
    testUnsuccessful : struct_PhaseAlgoritm;
    fb_pnsOn : fb_ph_Switch;
    fb_LowOil : fb_ph_WaitAnalogValue;
    fb_BreakPuskTimer_Poil : fb_ph_Timer;
    fb_Poil_DefenseActive : fb_ph_CustomPhase;
    fb_nuOn : fb_ph_CustomPhase;
    fb_nu1On : fb_ph_OilPump;
    fb_nu2On : fb_ph_OilPump;
    fb_autoNuOn : fb_ph_algoritm;
    fb_di_dPmg : fb_ph_CustomPhase;
    fb_dP_oilGas100 : fb_ph_WaitAnalogValue;
    fb_runProtect_dP : fb_ph_CustomPhase;
    fb_testUnsuccessful : fb_ph_CustomPhase;
    _sunpackerCommand : fb_sunpackerCommand;
    _statusAi : TYPE_StatusAi;
    _Answers : TYPE_Answers;
    _statusDualInput : TYPE_statusDualInput;
    _DualStateImAction : TYPE_DualStateImAction;
    _PhaseAlgoritmAction : TYPE_PhaseAlgoritmAction;
    source : BYTE;
    cmd : BYTE;
    lastCmd : BYTE;
    source_for_Status : BYTE;
    cmd_for_Status : BYTE;
    command_error_for_Status : BYTE;
    resetCmdTimer : TON;
    resetCmdTimerPriznak : BOOL;
    onInit : BOOL;
    waitReset : TON;
  END_VAR
  VAR_EXTERNAL
    IM : ImConfig;
    algoritms : AlgoritmsConfig;
    ai : AiConfig;
    protections : ProtectionsConfig;
    AlgTimers : struct_AlgTimers;
  END_VAR

  IF NOT onInit THEN
                 fb_pnsOn(phaseNumber:=0, act:=_on);
                fb_LowOil(phaseNumber:=1);
   fb_BreakPuskTimer_Poil(phaseNumber:=3, delay:=T#240S);
    fb_Poil_DefenseActive(phaseNumber:=5);
                  fb_nuOn(phaseNumber:=6);
                 fb_nu1On(phaseNumber:=11, act:=_on);
                 fb_nu2On(phaseNumber:=12, act:=_on);
              fb_autoNuOn(phaseNumber:=7, act:=_run, waitCompletion:=FALSE);
               fb_di_dPmg(phaseNumber:=8);
          fb_dP_oilGas100(phaseNumber:=9);
         fb_runProtect_dP(phaseNumber:=10);
      fb_testUnsuccessful(phaseNumber:=17);

  onInit:=TRUE;
  END_IF;

                fb_pnsOn(StrPh:=pnsOn, Im:=IM.pns);
               fb_LowOil(StrPh:=LowOil, ai:=ai.Davlenie_masla_smazki_nizkoe, more:=im.AutoPns_UstRun.Value);
  fb_BreakPuskTimer_Poil(StrPh:=BreakPuskTimer_Poil, timer:=AlgTimers.puskOilSystem_BreakPuskTimer_Poil);
   fb_Poil_DefenseActive(StrPh:=Poil_DefenseActive);
                 fb_nuOn(StrPh:=nuOn);
                fb_nu1On(StrPh:=nu1On, Im:=Im.nu1);
                fb_nu2On(StrPh:=nu2On, Im:=Im.nu2);
             fb_autoNuOn(StrPh:=autoNuOn, alg:=algoritms.autoNu);
              fb_di_dPmg(StrPh:=di_dPmg);
         fb_dP_oilGas100(StrPh:=dP_oilGas100, ai:=ai.Perepad_davleniya_maslo_gaz, more:=im.PuskOilSystem_UstdPmg.Value);
        fb_runProtect_dP(StrPh:=runProtect_dP);
     fb_testUnsuccessful(StrPh:=testUnsuccessful);

  IF StrAlg.isRuning THEN

      StrAlg.hasError := LowOil.error OR dP_oilGas100.error OR pnsOn.error OR testUnsuccessful.error;

      IF pnsOn.top THEN
          runPhase(LowOil);
      END_IF;

      IF LowOil.top THEN
          runAiProtection(protections.Davlenie_masla_smazki_nizkoe_LA);
          runPhase(Poil_DefenseActive);

          ai.Davlenie_masla_smazki_nizkoe.Disabled_LA:=FALSE;
          ai.Davlenie_masla_smazki_nizkoe.Disabled_LW:=FALSE;
          ai.Davlenie_masla_smazki_visokoe.Disabled_LW:=FALSE;
      END_IF;

      IF Poil_DefenseActive.start AND NOT Poil_DefenseActive.top THEN
         Poil_DefenseActive.top:=protections.Davlenie_masla_smazki_nizkoe_LA.isRunning;
      END_IF;

      IF Poil_DefenseActive.top THEN
         (* runPhase(autoNuOn);*)
  	runPhase(nuOn);
      END_IF;

      IF nuOn.start AND NOT nuOn.top THEN
          IF IM.AutoNU_mainNU.Value = 0 THEN
              runPhase(nu1On);
          END_IF;

          IF IM.AutoNU_mainNU.Value = 1 THEN
              runPhase(nu2On);
          END_IF;
         nuOn.top:= Im.nu1.onStatus = _statusDualInput.STATUS_ON OR Im.nu2.onStatus = _statusDualInput.STATUS_ON;
      END_IF;

      IF nuOn.top THEN
  	runPhase(di_dPmg);
            runPhase(dP_oilGas100);
      END_IF;

      IF di_dPmg.start AND NOT di_dPmg.top THEN
         di_dPmg.top:= NOT IM.SingleSignals.dP_maslo_gaz_menshe_100_kPa.Q;
      END_IF;

      IF dP_oilGas100.top AND di_dPmg.top THEN
            runPhase(autoNuOn);
  	runPhase(runProtect_dP);
  	runAiProtection(protections.Perepad_davleniya_maslo_gaz_LA);
            runDiProtection(protections.dP_maslo_gaz_menshe_100_kPa_DI);
            ai.Perepad_davleniya_maslo_gaz.Disabled_LA:=FALSE;
            ai.Perepad_davleniya_maslo_gaz.Disabled_LW:=FALSE;
      END_IF;

      IF runProtect_dP.start AND NOT runProtect_dP.top THEN
         runProtect_dP.top:= protections.Perepad_davleniya_maslo_gaz_LA.isRunning AND protections.dP_maslo_gaz_menshe_100_kPa_DI.isRunning;
      END_IF;

      IF BreakPuskTimer_Poil.top AND (NOT runProtect_dP.top) THEN
  	testUnsuccessful.error:=TRUE;
      END_IF;

      IF runProtect_dP.top THEN
            resetPhase(BreakPuskTimer_Poil);
  	waitReset(IN:=TRUE);
      END_IF;

      IF waitReset.Q AND NOT (algoritms.Apusk.isRuning OR algoritms.SemiAutoPusk.isRuning) THEN
      resetAndDisable(StrAlg);
      END_IF;

      StrAlg.isEnded:=runProtect_dP.top;
  END_IF;

  StrAlg.CanRun := StrAlg.inCanRun;
  StrAlg.OpcCommandsDisabled := StrAlg.inOpcCommandsDisabled;

  (* ---- Если управление с ВУ заблокировано, то  передаем команду из алгоритма ---- *)
  IF StrAlg.inOpcCommandsDisabled THEN
  	StrAlg.inCommand := StrAlg.inCommand_Alg;
  ELSE (* иначе передаем команду с АРМа*)
  	StrAlg.inCommand := StrAlg.inCommand_ARM;
  END_IF;

  _sunpackerCommand(command := StrAlg.inCommand);
  	source := _sunpackerCommand.source;
  	cmd := _sunpackerCommand.cmd;

  IF cmd <> 0 AND lastCmd <> cmd AND (((NOT StrAlg.opcCommandsDisabled) AND source > 0) OR source = 0) then
  	CASE BYTE_TO_INT(cmd) OF
  		(*cmdRun*) 1: 	IF (StrAlg.CanRun) THEN
  					StrAlg.isRuning := TRUE;
  					StrAlg.isEnded := FALSE;
  					StrAlg.hasError := FALSE;
  					(*****************       OnRun       *****************)
                                                    runPhase(pnsOn);
                                                    runPhase(BreakPuskTimer_Poil);
                                                    runPhase(testUnsuccessful);
  					cmd_for_Status := cmd;
  					source_for_Status := source;
  					command_error_for_Status := 0;
  				ELSE
  					StrAlg.isRuning := FALSE;
  					StrAlg.isEnded := FALSE;
  					StrAlg.hasError 	:= FALSE;

  					cmd_for_Status := 0;
  					source_for_Status := source;
  					command_error_for_Status := cmd;
  				END_IF;
  		(*cmdReset*) 2: 	StrAlg.isRuning := FALSE;
  				StrAlg.isEnded := FALSE;
  				StrAlg.hasError 	:= FALSE;

                                           (*****************       OnReset       *****************)
                                          waitReset(IN:=FALSE);
                                          resetPhase(pnsOn);
                                          resetPhase(LowOil);
                                          resetPhase(BreakPuskTimer_Poil);
                                          resetPhase(Poil_DefenseActive);
                                          resetPhase(autoNuOn);
                                          resetPhase(nu1On);
                                          resetPhase(nu2On);
                                          resetPhase(nuOn);
                                          resetPhase(di_dPmg);
                                          resetPhase(dP_oilGas100);
                                          resetPhase(runProtect_dP);
                                          resetPhase(testUnsuccessful);
  	                              (*protections.P_masla_smazki_nizkoe_LA.inOpcCommandsDisabled:=FALSE;
                                          protections.DavlenieMaslaSmazkiDi.inOpcCommandsDisabled:=FALSE;
                                          protections.dP_maslogaz_LA.inOpcCommandsDisabled:=FALSE;
                                          protections.dP_masloGaz_LowDI.inOpcCommandsDisabled:=FALSE;*)

  				cmd_for_Status := cmd;
  				source_for_Status := source;
  				command_error_for_Status := 0;
  	END_CASE;
  	resetCmdTimer(IN := false);
  	resetCmdTimerPriznak := TRUE;
  END_IF;
  lastCmd := cmd;

  resetCmdTimer(IN := resetCmdTimerPriznak, PT := T#5S);
  IF resetCmdTimer.Q THEN
  	resetCmdTimerPriznak := FALSE;
  	source_for_Status := 0;
  	cmd_for_Status := 0;
  	command_error_for_Status := 0;
  END_IF;

  StrAlg.Start:= pnsOn.startStatus
              OR LowOil.startStatus
              OR BreakPuskTimer_Poil.startStatus
              OR Poil_DefenseActive.startStatus
              OR nuOn.startStatus
              OR di_dPmg.startStatus
              OR dP_oilGas100.startStatus
              OR runProtect_dP.startStatus
              OR testUnsuccessful.startStatus;

  StrAlg.Error:= pnsOn.errorStatus
              OR LowOil.errorStatus
              OR BreakPuskTimer_Poil.errorStatus
              OR Poil_DefenseActive.errorStatus
              OR nuOn.errorStatus
              OR di_dPmg.errorStatus
              OR dP_oilGas100.errorStatus
              OR runProtect_dP.errorStatus
              OR testUnsuccessful.errorStatus;

  StrAlg.Top:=   pnsOn.topStatus
              OR LowOil.topStatus
              OR BreakPuskTimer_Poil.topStatus
              OR Poil_DefenseActive.topStatus
              OR nuOn.topStatus
              OR di_dPmg.topStatus
              OR dP_oilGas100.topStatus
              OR runProtect_dP.topStatus
              OR testUnsuccessful.topStatus;

  (*TODO: TYPE PROGRAM CODE HERE*)
  StrAlg.status :=  SHL(BYTE_TO_DWORD(source_for_Status), 29)
  			OR SHL(BYTE_TO_DWORD(cmd_for_Status), 26)
  			OR SHL(BYTE_TO_DWORD(command_error_for_Status), 23)
  			OR SHL(BOOL_TO_DWORD(StrAlg.OpcCommandsDisabled ), 21)
  			OR SHL(BOOL_TO_DWORD(StrAlg.hasError),4)
  			OR SHL(BOOL_TO_DWORD(StrAlg.CanRun),2)
  			OR SHL(BOOL_TO_DWORD(StrAlg.isEnded),1)
  			OR BOOL_TO_DWORD(StrAlg.isRuning);
END_FUNCTION_BLOCK

FUNCTION_BLOCK fb_singleOutput
  VAR_IN_OUT
    signal : BOOL;
    str_SO : struct_singleOutput;
  END_VAR
  VAR
    pulseTimer : TON;
    resetCmdTimer : TON;
    TON_Command : TON;
    source : BYTE;
    cmd : BYTE;
    lastCmd : BYTE;
    source_for_Status : BYTE;
    cmd_for_Status : BYTE;
    command_error_for_Status : BYTE;
    pulseTimerPriznak : BOOL;
    resetCmdTimerPriznak : BOOL;
    _sunpackerCommand : fb_sunpackerCommand;
  END_VAR

  str_SO.OpcCommandsDisabled := str_SO.inOpcCommandsDisabled;

  (* ---- Если управление с ВУ заблокировано, то передаем команду из алгоритма ---- *)
  IF str_SO.inOpcCommandsDisabled THEN
  	str_SO.inCommand := str_SO.inCommand_Alg;
  ELSE (* иначе передаем команду с АРМа*)
  	str_SO.inCommand := str_SO.inCommand_ARM;
  END_IF;

  (*Распаковка команды*)
  _sunpackerCommand(command := str_SO.inCommand);
  	cmd := _sunpackerCommand.cmd;
  	source := _sunpackerCommand.source;

  (*Обработка команды*)
  IF cmd <> 0 AND lastCmd <> cmd and (((NOT str_SO.OpcCommandsDisabled) AND source > 0) OR source = 0) then
  	CASE BYTE_TO_INT(cmd) OF
  	(*cmd_on*) 1 :
  			str_SO.Q := TRUE;
  			pulseTimer(IN := FALSE);
  			pulseTimerPriznak := FALSE;
  			resetCmdTimer(IN := FALSE);
  			resetCmdTimerPriznak := TRUE;
  	(*cmd_off*) 2 :
  			str_SO.Q := FALSE;
  			pulseTimer(IN := FALSE);
  			pulseTimerPriznak := FALSE;
  			resetCmdTimer(IN := FALSE);
  			resetCmdTimerPriznak := TRUE;
  	(*cmd_pulse*) 3 :
  			str_SO.Q := TRUE;
                                pulseTimer(IN := FALSE);
                                pulseTimerPriznak := TRUE;
  			resetCmdTimer(IN := FALSE);
                                resetCmdTimerPriznak := FALSE;
  	END_CASE;
  	source_for_Status := source;
  	cmd_for_Status := cmd;
  	command_error_for_Status := 0;
  END_IF;
  lastCmd := cmd;

  pulseTimer(IN := pulseTimerPriznak, PT := str_SO.wait_time);
  pulseTimer();
  IF pulseTimer.Q THEN
  	pulseTimer(IN := FALSE);
  	pulseTimerPriznak := FALSE;

  	str_SO.Q := FALSE;

  	source_for_Status := 0;
  	cmd_for_Status := 0;
  	command_error_for_Status := 0;
  END_IF;

  resetCmdTimer(IN := resetCmdTimerPriznak, PT := T#10S);
  resetCmdTimer();
  IF resetCmdTimer.Q THEN
  	resetCmdTimer(IN := FALSE);
  	resetCmdTimerPriznak := FALSE;

  	source_for_Status := 0;
  	cmd_for_Status := 0;
  	command_error_for_Status := 0;
  END_IF;

  signal:= str_SO.Q;

  (*TON_Command(IN:= (inCommand <> 0) AND (source = 0), PT:= T#2S);*)
      (*IF TON_Command.Q THEN*)
          (*inCommand := 0;*)
      (*END_IF;*)
  str_SO.status :=                           shl(BYTE_TO_DWORD(source_for_Status), 29)
  				OR shl(BYTE_TO_DWORD(cmd_for_Status), 26)
  				OR shl(BYTE_TO_DWORD(command_error_for_Status), 23)
  				OR shl(BOOL_TO_DWORD(str_SO.OpcCommandsDisabled), 21)
  				OR BOOL_TO_DWORD(str_SO.Q);
END_FUNCTION_BLOCK

FUNCTION_BLOCK fb_singleOutput_Init
  VAR_INPUT
    data_Ini : BOOL;
    inOpcCommandsDisabled : BOOL;
    wait_time : TIME;
  END_VAR
  VAR_IN_OUT
    str_SO : struct_singleOutput;
  END_VAR
  VAR_OUTPUT
    Init : BOOL         := FALSE;
  END_VAR

  (*****            Функциональный блок переинициализации структуры  singleOutput          *****)

  Init := FALSE;

      IF data_Ini THEN                            (* Параметрам требуется переинициализация. *)
          str_SO.inOpcCommandsDisabled    := inOpcCommandsDisabled;
          str_SO.wait_time                := wait_time;

           data_Ini:=FALSE;
          Init := TRUE;
      END_IF;
   IF Init THEN
          inOpcCommandsDisabled := FALSE;
          wait_time := T#0S;
     END_IF;
END_FUNCTION_BLOCK

FUNCTION_BLOCK fb_singleSignal
  VAR_INPUT
    signal : TYPE_ReliableBit;
  END_VAR
  VAR_IN_OUT
    str_SS : struct_singleSignal;
  END_VAR
  VAR
    TimerOn : TON;
    TimerOff : TOF;
  END_VAR

  str_SS.reliability:=signal.reliability;

  IF NOT str_SS.inverse THEN
  TimerOn(IN:=(signal.value AND str_SS.reliability AND NOT str_SS.Disabled_Sig), PT:=str_SS.DelayOn);
  ELSE
  TimerOn(IN:=(signal._inversed AND str_SS.reliability AND NOT str_SS.Disabled_Sig), PT:=str_SS.DelayOn);
  END_IF;

  TimerOff(IN:=TimerOn.Q, PT:=str_SS.DelayOff);

  str_SS.Q:=TimerOff.Q;

  str_SS.status:= SHL(BOOL_TO_DWORD(NOT str_SS.reliability), 15)
  	OR BOOL_TO_DWORD(str_SS.Q);
END_FUNCTION_BLOCK

FUNCTION_BLOCK fb_singleSignal_Init
  VAR_INPUT
    data_Ini : BOOL;
    inverse : BOOL;
    DelayOn : TIME;
    DelayOff : TIME;
  END_VAR
  VAR_IN_OUT
    str_SS : struct_singleSignal;
  END_VAR
  VAR_OUTPUT
    Init : BOOL         := FALSE;
  END_VAR

  (*****            Функциональный блок переинициализации структуры  singleSignal          *****)
  Init := FALSE;

      IF data_Ini THEN                            (* Параметрам требуется переинициализация. *)
          str_SS.inverse                := inverse;
          str_SS.DelayOn                := DelayOn;
          str_SS.DelayOff               := DelayOff;

          data_Ini:=FALSE;
          Init := TRUE;
      END_IF;
   IF Init THEN
          inverse := FALSE;
          DelayOn := T#0S;
          DelayOff:= T#0S;
   END_IF;
END_FUNCTION_BLOCK

FUNCTION_BLOCK fb_vibegPNSAlg
  VAR_IN_OUT
    StrAlg : struct_Alg;
  END_VAR
  VAR
    autoPnsOff : struct_PhaseAlgoritm;
    waitVibeg : struct_PhaseAlgoritm;
    pnsOff : struct_PhaseAlgoritm;
    vibegEnd : struct_PhaseAlgoritm;
  END_VAR
  VAR_IN_OUT
    algContinue : struct_Question;
  END_VAR
  VAR
    fb_autoPnsOff : fb_ph_algoritm;
    fb_waitVibeg : fb_ph_Timer;
    fb_algContinue : fb_Question;
    fb_pnsOff : fb_ph_Switch;
    fb_vibegEnd : fb_ph_CustomPhase;
    _sunpackerCommand : fb_sunpackerCommand;
    _statusAi : TYPE_StatusAi;
    _Answers : TYPE_Answers;
    _statusDualInput : TYPE_statusDualInput;
    _DualStateImAction : TYPE_DualStateImAction;
    _PhaseAlgoritmAction : TYPE_PhaseAlgoritmAction;
    source : BYTE;
    cmd : BYTE;
    lastCmd : BYTE;
    source_for_Status : BYTE;
    cmd_for_Status : BYTE;
    command_error_for_Status : BYTE;
    resetCmdTimer : TON;
    resetCmdTimerPriznak : BOOL;
    onInit : BOOL;
    waitReset : TON;
  END_VAR
  VAR_EXTERNAL
    IM : ImConfig;
    algoritms : AlgoritmsConfig;
    ai : AiConfig;
    protections : ProtectionsConfig;
    AlgTimers : struct_AlgTimers;
  END_VAR

  IF NOT onInit THEN
   fb_autoPnsOff(phaseNumber:=0, act:=_reset, waitCompletion:=FALSE);
    fb_waitVibeg(phaseNumber:=1, delay:=T#30S);
       algContinue.AnswerVariants:=_Answers.ANS_YES;
       fb_pnsOff(phaseNumber:=2, act:=_off);
     fb_vibegEnd(phaseNumber:=14);
  onInit:=TRUE;
  END_IF;

   fb_autoPnsOff(StrPh:=autoPnsOff, alg:=algoritms.autoPns);
    fb_waitVibeg(StrPh:=waitVibeg, timer:=AlgTimers.vibegPNS_Timer);
  fb_algContinue(StrQ:=algContinue);
       fb_pnsOff(StrPh:=pnsOff, Im:=IM.pns);
     fb_vibegEnd(StrPh:=vibegEnd);

  IF StrAlg.isRuning THEN

  StrAlg.hasError := autoPnsOff.error OR pnsOff.error;

      IF IM.pns.onStatus = _statusDualInput.STATUS_ON AND NOT vibegEnd.top THEN

  	runPhase(vibegEnd);
            runPhase(waitVibeg);
            askQuestion(algContinue);

      END_IF;

      IF waitVibeg.top OR (algContinue.answer = _Answers.ANS_YES) THEN
  	vibegEnd.top:=TRUE;
  	resetPhase(waitVibeg);
            resetQuestion(algContinue);

            resetAiProtection(protections.Davlenie_masla_smazki_nizkoe_LA);

  	ai.Davlenie_masla_smazki_nizkoe.Disabled_LA:=TRUE;
            ai.Davlenie_masla_smazki_nizkoe.Disabled_LW:=TRUE;
            ai.Davlenie_masla_smazki_visokoe.Disabled_LW:=TRUE;
  	runPhase(pnsOff);
      END_IF;

      StrAlg.isEnded:=pnsOff.top;

  END_IF;

  StrAlg.CanRun := StrAlg.inCanRun;
  StrAlg.OpcCommandsDisabled := StrAlg.inOpcCommandsDisabled;

  (* ---- Если управление с ВУ заблокировано, то  передаем команду из алгоритма ---- *)
  IF StrAlg.inOpcCommandsDisabled THEN
  	StrAlg.inCommand := StrAlg.inCommand_Alg;
  ELSE (* иначе передаем команду с АРМа*)
  	StrAlg.inCommand := StrAlg.inCommand_ARM;
  END_IF;

  _sunpackerCommand(command := StrAlg.inCommand);
  	source := _sunpackerCommand.source;
  	cmd := _sunpackerCommand.cmd;

  IF cmd <> 0 AND lastCmd <> cmd AND (((NOT StrAlg.opcCommandsDisabled) AND source > 0) OR source = 0) then
  	CASE BYTE_TO_INT(cmd) OF
  		(*cmdRun*) 1: 	IF (StrAlg.CanRun) THEN
  					StrAlg.isRuning := TRUE;
  					StrAlg.isEnded := FALSE;
  					StrAlg.hasError := FALSE;
  					(*****************       OnRun       *****************)
                                                    runPhase(autoPnsOff);

  					cmd_for_Status := cmd;
  					source_for_Status := source;
  					command_error_for_Status := 0;
  				ELSE
  					StrAlg.isRuning := FALSE;
  					StrAlg.isEnded := FALSE;
  					StrAlg.hasError 	:= FALSE;

  					cmd_for_Status := 0;
  					source_for_Status := source;
  					command_error_for_Status := cmd;
  				END_IF;
  		(*cmdReset*) 2: 	StrAlg.isRuning := FALSE;
  				StrAlg.isEnded := FALSE;
  				StrAlg.hasError 	:= FALSE;

                                           (*****************       OnReset       *****************)
                                         waitReset(IN:=FALSE);
                                         resetPhase(autoPnsOff);
                                         resetPhase(waitVibeg);
                                         resetPhase(vibegEnd);
                                         resetPhase(pnsOff);
                                         resetQuestion(algContinue);

  				cmd_for_Status := cmd;
  				source_for_Status := source;
  				command_error_for_Status := 0;
  	END_CASE;
  	resetCmdTimer(IN := false);
  	resetCmdTimerPriznak := TRUE;
  END_IF;
  lastCmd := cmd;

  resetCmdTimer(IN := resetCmdTimerPriznak, PT := T#5S);
  IF resetCmdTimer.Q THEN
  	resetCmdTimerPriznak := FALSE;
  	source_for_Status := 0;
  	cmd_for_Status := 0;
  	command_error_for_Status := 0;
  END_IF;

  StrAlg.Start:= autoPnsOff.startStatus
              OR waitVibeg.startStatus
              OR pnsOff.startStatus
              OR vibegEnd.startStatus;

  StrAlg.Error:= autoPnsOff.errorStatus
              OR waitVibeg.errorStatus
              OR pnsOff.errorStatus
              OR vibegEnd.errorStatus;

  StrAlg.Top:=   autoPnsOff.topStatus
              OR waitVibeg.topStatus
              OR pnsOff.topStatus
              OR vibegEnd.topStatus;

  (*TODO: TYPE PROGRAM CODE HERE*)
  StrAlg.status :=  SHL(BYTE_TO_DWORD(source_for_Status), 29)
  			OR SHL(BYTE_TO_DWORD(cmd_for_Status), 26)
  			OR SHL(BYTE_TO_DWORD(command_error_for_Status), 23)
  			OR SHL(BOOL_TO_DWORD(StrAlg.OpcCommandsDisabled ), 21)
  			OR SHL(BOOL_TO_DWORD(StrAlg.hasError),4)
  			OR SHL(BOOL_TO_DWORD(StrAlg.CanRun),2)
  			OR SHL(BOOL_TO_DWORD(StrAlg.isEnded),1)
  			OR BOOL_TO_DWORD(StrAlg.isRuning);
END_FUNCTION_BLOCK

FUNCTION_BLOCK fillingAlg
  VAR_IN_OUT
    StrAlg : struct_Alg;
  END_VAR
  VAR
    BreakPuskTimer : struct_PhaseAlgoritm;
    kran3bOpen : struct_PhaseAlgoritm;
    kran4Open : struct_PhaseAlgoritm;
    waitAfterKran4 : struct_PhaseAlgoritm;
    kran5Close : struct_PhaseAlgoritm;
    didPKran1 : struct_PhaseAlgoritm;
    kran1Open : struct_PhaseAlgoritm;
    kran2Open : struct_PhaseAlgoritm;
    kran3bClose : struct_PhaseAlgoritm;
    kran4Close : struct_PhaseAlgoritm;
    RunProtection_kr1 : struct_PhaseAlgoritm;
    RunProtection_kr2 : struct_PhaseAlgoritm;
    waitAfterKran5 : struct_PhaseAlgoritm;
    testUnsuccessfulFilling : struct_PhaseAlgoritm;
    fb_BreakPuskTimer : fb_ph_Timer;
    fb_kran3bOpen : fb_ph_Kran;
    fb_kran4Open : fb_ph_Kran;
    fb_waitAfterKran4 : fb_ph_Timer;
    fb_kran5Close : fb_ph_Kran;
    fb_didPKran1 : fb_ph_CustomPhase;
    fb_kran1Open : fb_ph_Kran;
    fb_kran2Open : fb_ph_Kran;
    fb_kran3bClose : fb_ph_Kran;
    fb_kran4Close : fb_ph_Kran;
    fb_RunProtection_kr1 : fb_ph_DIprotection;
    fb_RunProtection_kr2 : fb_ph_DIprotection;
    fb_waitAfterKran5 : fb_ph_Timer;
    fb_testUnsuccessfulFilling : fb_ph_CustomPhase;
    _sunpackerCommand : fb_sunpackerCommand;
    _DualStateImAction : TYPE_DualStateImAction;
    _PhaseAlgoritmAction : TYPE_PhaseAlgoritmAction;
    source : BYTE;
    cmd : BYTE;
    lastCmd : BYTE;
    source_for_Status : BYTE;
    cmd_for_Status : BYTE;
    command_error_for_Status : BYTE;
    resetCmdTimer : TON;
    resetCmdTimerPriznak : BOOL;
    onInit : BOOL;
    waitReset : TON;
  END_VAR
  VAR_EXTERNAL
    IM : ImConfig;
    ai : AiConfig;
    protections : ProtectionsConfig;
    AlgTimers : struct_AlgTimers;
    algoritms : AlgoritmsConfig;
  END_VAR

  IF NOT onInit THEN

           fb_BreakPuskTimer(phaseNumber:=0, delay:=T#240S);
               fb_kran3bOpen(phaseNumber:=1, act:=_on);
                fb_kran4Open(phaseNumber:=2, act:=_on);
           fb_waitAfterKran4(phaseNumber:=3, delay:=T#10S);
               fb_kran5Close(phaseNumber:=4, act:=_off);
                fb_didPKran1(phaseNumber:=5);
                fb_kran1Open(phaseNumber:=7, act:=_on);
                fb_kran2Open(phaseNumber:=8, act:=_on);
              fb_kran3bClose(phaseNumber:=9, act:=_off);
               fb_kran4Close(phaseNumber:=10, act:=_off);
        fb_RunProtection_kr1(phaseNumber:=11, act:=_run);
        fb_RunProtection_kr2(phaseNumber:=12, act:=_run);
           fb_waitAfterKran5(phaseNumber:=13, delay:=T#60S);
  fb_testUnsuccessfulFilling(phaseNumber:=17);

  onInit:=TRUE;
  END_IF;

           fb_BreakPuskTimer(StrPh:=BreakPuskTimer, timer:=AlgTimers.filling_BreakPuskTimer);
               fb_kran3bOpen(StrPh:=kran3bOpen, Im:=Im.kran3b);
                fb_kran4Open(StrPh:=kran4Open, Im:=Im.kran4);
           fb_waitAfterKran4(StrPh:=waitAfterKran4, timer:=AlgTimers.filling_waitAfterKran4);
               fb_kran5Close(StrPh:=kran5Close, Im:=Im.kran5);
                fb_didPKran1(StrPh:=didPKran1);
                fb_kran1Open(StrPh:=kran1Open, Im:=Im.kran1);
                fb_kran2Open(StrPh:=kran2Open, Im:=Im.kran2);
              fb_kran3bClose(StrPh:=kran3bClose, Im:=Im.kran3b);
               fb_kran4Close(StrPh:=kran4Close, Im:=Im.kran4);
        fb_RunProtection_kr1(StrPh:=RunProtection_kr1 , StrDiP:=protections.Kran1sdvig);
        fb_RunProtection_kr2(StrPh:=RunProtection_kr2 , StrDiP:=protections.Kran2sdvig);
           fb_waitAfterKran5(StrPh:=waitAfterKran5, timer:=AlgTimers.filling_waitAfterKran5);
  fb_testUnsuccessfulFilling(StrPh:=testUnsuccessfulFilling);

  StrAlg.CanRun := StrAlg.inCanRun;
  StrAlg.OpcCommandsDisabled := StrAlg.inOpcCommandsDisabled;

  IF StrAlg.isRuning THEN

      StrAlg.hasError := kran3bOpen.error OR kran4Open.error OR kran5Close.error OR kran5Close.error
      OR kran1Open.error OR kran2Open.error OR kran3bClose.error OR kran4Close.error OR testUnsuccessfulFilling.error;

      IF kran4Open.top THEN
          runPhase(waitAfterKran4);
      END_IF;

      IF waitAfterKran4.top THEN
          runPhase(kran5Close);
      END_IF;

      IF kran3bOpen.top AND kran5Close.top THEN
         runPhase(waitAfterKran5);
         runPhase(didPKran1);
      END_IF;

      IF didPKran1.start AND NOT didPKran1.top THEN
      didPKran1.top:= im.singleSignals.dP_gaza_kr_1.Q;
      END_IF;

      IF waitAfterKran5.top AND didPKran1.top THEN
            runPhase(kran1Open);
  	runPhase(kran2Open);
      END_IF;

      IF kran1Open.top AND kran2Open.top THEN
            runPhase(kran4Close);
  	runPhase(kran3bClose);
      END_IF;

      IF kran4Close.top AND kran3bClose.top THEN

            runPhase(RunProtection_kr1);
            runPhase(RunProtection_kr2);

            runAiProtection(protections.Vibroskorost_OP_ED_t1_HA);
            runAiProtection(protections.Vibroskorost_OYP_ED_so_storony_redyctora_t2_HA);
            runAiProtection(protections.Vibroskorost_OYP_kolesa_ED_t3_HA);
            runAiProtection(protections.Vibroskorost_OP_shesterni_nagnetatelya_t6_HA);

      END_IF;

      IF BreakPuskTimer.top AND NOT (RunProtection_kr1.top AND RunProtection_kr2.top ) THEN
  	testUnsuccessfulFilling.error:=TRUE;
      END_IF;

      IF RunProtection_kr1.top AND RunProtection_kr2.top THEN
            resetPhase(BreakPuskTimer);
  	waitReset(IN:=TRUE, PT:= T#2S);
      END_IF;

      IF waitReset.Q AND NOT (algoritms.Apusk.isRuning OR algoritms.SemiAutoPusk.isRuning) THEN
  	resetIfRunning(StrAlg);
      END_IF;

      StrAlg.isEnded:= RunProtection_kr1.top AND RunProtection_kr2.top;
  END_IF;

  StrAlg.CanRun := StrAlg.inCanRun;
  StrAlg.OpcCommandsDisabled := StrAlg.inOpcCommandsDisabled;

  (* ---- Если управление с ВУ заблокировано, то  передаем команду из алгоритма ---- *)
  IF StrAlg.inOpcCommandsDisabled THEN
  	StrAlg.inCommand := StrAlg.inCommand_Alg;
  ELSE (* иначе передаем команду с АРМа*)
  	StrAlg.inCommand := StrAlg.inCommand_ARM;
  END_IF;

  _sunpackerCommand(command := StrAlg.inCommand);
  	source := _sunpackerCommand.source;
  	cmd := _sunpackerCommand.cmd;

  IF cmd <> 0 AND lastCmd <> cmd AND (((NOT StrAlg.opcCommandsDisabled) AND source > 0) OR source = 0) then
  	CASE BYTE_TO_INT(cmd) OF
  		(*cmdRun*) 1: 	IF (StrAlg.CanRun) THEN
  					StrAlg.isRuning := TRUE;
  					StrAlg.isEnded := FALSE;
  					StrAlg.hasError := FALSE;
  					(*****************       OnRun       *****************)

                                                    runPhase(kran3bOpen);
                                                    runPhase(kran4Open);
                                                    runPhase(BreakPuskTimer);
                                                    runPhase(testUnsuccessfulFilling);

  					cmd_for_Status := cmd;
  					source_for_Status := source;
  					command_error_for_Status := 0;
  				ELSE
  					StrAlg.isRuning := FALSE;
  					StrAlg.isEnded := FALSE;
  					StrAlg.hasError 	:= FALSE;

  					cmd_for_Status := 0;
  					source_for_Status := source;
  					command_error_for_Status := cmd;
  				END_IF;
  		(*cmdReset*) 2: 	StrAlg.isRuning := FALSE;
  				StrAlg.isEnded := FALSE;
  				StrAlg.hasError 	:= FALSE;

                                           (*****************       OnReset       *****************)
                                          StrAlg.inCanRun:=FALSE;
                                          waitReset(IN:=FALSE);

                                          resetPhase(BreakPuskTimer);
                                          resetPhase(kran3bOpen);
                                          resetPhase(kran4Open);
                                          resetPhase(waitAfterKran4);
                                          resetPhase(kran5Close);
                                          resetPhase(didPKran1);
                                          resetPhase(kran1Open);
                                          resetPhase(kran2Open);
                                          resetPhase(kran3bClose);
                                          resetPhase(kran4Close);
  	                              resetPhase(RunProtection_kr1);
                                          resetPhase(RunProtection_kr2);
                                          resetPhase(waitAfterKran5);
                                          resetPhase(testUnsuccessfulFilling);

  				cmd_for_Status := cmd;
  				source_for_Status := source;
  				command_error_for_Status := 0;
  	END_CASE;
  	resetCmdTimer(IN := false);
  	resetCmdTimerPriznak := TRUE;
  END_IF;
  lastCmd := cmd;

  resetCmdTimer(IN := resetCmdTimerPriznak, PT := T#5S);
  IF resetCmdTimer.Q THEN
  	resetCmdTimerPriznak := FALSE;
  	source_for_Status := 0;
  	cmd_for_Status := 0;
  	command_error_for_Status := 0;
  END_IF;

  StrAlg.Start:= BreakPuskTimer.startStatus
              OR kran3bOpen.startStatus
              OR kran4Open.startStatus
              OR waitAfterKran4.startStatus
              OR kran5Close.startStatus
              OR didPKran1.startStatus
              OR kran1Open.startStatus
              OR kran2Open.startStatus
              OR kran3bClose.startStatus
              OR kran4Close.startStatus
              OR RunProtection_kr1.startStatus
              OR RunProtection_kr2.startStatus
              OR waitAfterKran5.startStatus
              OR testUnsuccessfulFilling.startStatus;

  StrAlg.Error:= BreakPuskTimer.errorStatus
              OR kran3bOpen.errorStatus
              OR kran4Open.errorStatus
              OR waitAfterKran4.errorStatus
              OR kran5Close.errorStatus
              OR didPKran1.errorStatus
              OR kran1Open.errorStatus
              OR kran2Open.errorStatus
              OR kran3bClose.errorStatus
              OR kran4Close.errorStatus
              OR RunProtection_kr1.errorStatus
              OR RunProtection_kr2.errorStatus
              OR waitAfterKran5.errorStatus
              OR testUnsuccessfulFilling.errorStatus;

  StrAlg.Top:=   BreakPuskTimer.topStatus
              OR kran3bOpen.topStatus
              OR kran4Open.topStatus
              OR waitAfterKran4.topStatus
              OR kran5Close.topStatus
              OR didPKran1.topStatus
              OR kran1Open.topStatus
              OR kran2Open.topStatus
              OR kran3bClose.topStatus
              OR kran4Close.topStatus
              OR RunProtection_kr1.topStatus
              OR RunProtection_kr2.topStatus
              OR waitAfterKran5.topStatus
              OR testUnsuccessfulFilling.topStatus;

  (*TODO: TYPE PROGRAM CODE HERE*)
  StrAlg.status :=  SHL(BYTE_TO_DWORD(source_for_Status), 29)
  			OR SHL(BYTE_TO_DWORD(cmd_for_Status), 26)
  			OR SHL(BYTE_TO_DWORD(command_error_for_Status), 23)
  			OR SHL(BOOL_TO_DWORD(StrAlg.OpcCommandsDisabled ), 21)
  			OR SHL(BOOL_TO_DWORD(StrAlg.hasError),4)
  			OR SHL(BOOL_TO_DWORD(StrAlg.CanRun),2)
  			OR SHL(BOOL_TO_DWORD(StrAlg.isEnded),1)
  			OR BOOL_TO_DWORD(StrAlg.isRuning);
END_FUNCTION_BLOCK

FUNCTION_BLOCK proc_AI
  VAR
    fb_T_medi_statora_faza_1 : fb_AiSourceMlp;
    fb_T_medi_statora_faza_2 : fb_AiSourceMlp;
    fb_T_medi_statora_faza_3 : fb_AiSourceMlp;
    fb_T_stali_statora_faza_1 : fb_AiSourceMlp;
    fb_T_stali_statora_faza_2 : fb_AiSourceMlp;
    fb_T_stali_statora_faza_3 : fb_AiSourceMlp;
    fb_T_goryachego_vozdyha_ed_t1 : fb_AiSourceMlp;
    fb_T_goryachego_vozdyha_ed_t2 : fb_AiSourceMlp;
    fb_T_holodnogo_vozdyha_ed_t1 : fb_AiSourceMlp;
    fb_T_holodnogo_vozdyha_ed_t2 : fb_AiSourceMlp;
    fb_T_OP_ED_t1 : fb_AiSourceMlp;
    fb_T_OYP_ED_so_storony_redyctora_t2 : fb_AiSourceMlp;
    fb_T_OYP_kolesa_ED_t3 : fb_AiSourceMlp;
    fb_T_OP_kolesa_nagnetatelya_t4 : fb_AiSourceMlp;
    fb_T_OP_shesterni_ED_t5 : fb_AiSourceMlp;
    fb_T_OP_redyctora_so_storony_nagnetatelya_t6 : fb_AiSourceMlp;
    fb_T_OYP_nagnetatelya_so_storony_redyctora_t7_1 : fb_AiSourceMlp;
    fb_T_OYP_nagnetatelya_so_storony_redyctora_t7_2 : fb_AiSourceMlp;
    fb_T_OYP_svobodnogo_konca_nagnetatelya_t8_1 : fb_AiSourceMlp;
    fb_T_OYP_svobodnogo_konca_nagnetatelya_t8_2 : fb_AiSourceMlp;
    fb_T_YP_rabochih_kolodok_nagnetatelya_t9 : fb_AiSourceMlp;
    fb_T_ne_rabochih_kolodok_YP_nagnetatelya_t10 : fb_AiSourceMlp;
    fb_T_gaz_in_nagnetatelia : fb_AiSourceMlp;
    fb_T_gaz_out_nagnetatelia : fb_AiSourceMlp;
    fb_T_masla_do_ABO : fb_AiSourceMlp;
    fb_T_masla_posle_ABO : fb_AiSourceMlp;
    fb_T_masla_v_maslobake : fb_AiSourceMlp;
    fb_T_masla_v_maslobake_nad_ten : fb_AiSourceMlp;
    fb_T_naryjnogo_vozdyxa : fb_AiSourceMlp;
    fb_T_vozduha_V_shkaf : fb_AiSourceMlp;
    fb_Davlenie_impylsnogo_gaza : fb_AiSourceMlp;
    fb_Yroven_masla_v_maslobake : fb_AiSourceMlp;
    fb_Osevoi_sdvig_nagnetatelya_vpravo : fb_AiSourceMlp;
    fb_Osevoi_sdvig_nagnetatelya_vlevo : fb_AiSourceMlp;
    fb_Tok_statora : fb_AiSourceMlp;
    fb_Kontrol_220_perem : fb_AiSourceMlp;
    fb_Kontrol_220_post : fb_AiSourceMlp;
    fb_Davlenie_gaza_na_vhode_nagnetatelya : fb_AiSourceMlp;
    fb_Davlenie_gaza_na_vihode_nagnetatelya : fb_AiSourceMlp;
    fb_Perepad_davleniya_maslo_gaz : fb_AiSourceMlp;
    fb_Davlenie_masla_posle_nasosa_yplotneniya : fb_AiSourceMlp;
    fb_Davlenie_masla_smazki_nizkoe : fb_AiSourceMlp;
    fb_Davlenie_masla_smazki_visokoe : fb_AiSourceMlp;
    fb_Davlenie_masla_smazki_posle_GNS : fb_AiSourceMlp;
    fb_Perepad_davleniya_gaza_na_konfyzore : fb_AiSourceMlp;
    fb_Perepad_davleniya_masla_na_maslyanom_filtre : fb_AiSourceMlp;
    fb_Vibroskorost_OP_ED_t1 : fb_AiSourceMlp;
    fb_Vibroskorost_OYP_ED_so_storony_redyctora_t2 : fb_AiSourceMlp;
    fb_Vibroskorost_OYP_kolesa_ED_t3 : fb_AiSourceMlp;
    fb_Vibroskorost_OP_kolesa_nagnetatelya_t4 : fb_AiSourceMlp;
    fb_Vibroskorost_OP_shesterni_ED_t5 : fb_AiSourceMlp;
    fb_Vibroskorost_OP_shesterni_nagnetatelya_t6 : fb_AiSourceMlp;
  END_VAR
  VAR_EXTERNAL
    ai : AiConfig;
    arAIN_0 : TItemAIN;
    arAIN_1 : TItemAIN;
    arAIN_2 : TItemAIN;
    arAIN_3 : TItemAIN;
    arAIN_4 : TItemAIN;
    arAIN_5 : TItemAIN;
    arAIN_6 : TItemAIN;
    arAIN_7 : TItemAIN;
    arAIN_8 : TItemAIN;
    arAIN_9 : TItemAIN;
    arAIN_10 : TItemAIN;
    arAIN_11 : TItemAIN;
    arAIN_12 : TItemAIN;
    arAIN_13 : TItemAIN;
    arAIN_14 : TItemAIN;
    arAIN_15 : TItemAIN;
    arAIN_16 : TItemAIN;
    arAIN_17 : TItemAIN;
    arAIN_18 : TItemAIN;
    arAIN_19 : TItemAIN;
    arAIN_20 : TItemAIN;
    arAIN_21 : TItemAIN;
    arAIN_22 : TItemAIN;
    arAIN_23 : TItemAIN;
    arAIN_24 : TItemAIN;
    arAIN_25 : TItemAIN;
    arAIN_26 : TItemAIN;
    arAIN_27 : TItemAIN;
    arAIN_28 : TItemAIN;
    arAIN_29 : TItemAIN;
    arAIN_30 : TItemAIN;
    arAIN_31 : TItemAIN;
    arAIN_32 : TItemAIN;
    arAIN_33 : TItemAIN;
    arAIN_34 : TItemAIN;
    arAIN_35 : TItemAIN;
    arAIN_36 : TItemAIN;
    arAIN_37 : TItemAIN;
    arAIN_38 : TItemAIN;
    arAIN_39 : TItemAIN;
    arAIN_40 : TItemAIN;
    arAIN_41 : TItemAIN;
    arAIN_42 : TItemAIN;
    arAIN_43 : TItemAIN;
    arAIN_44 : TItemAIN;
    arAIN_45 : TItemAIN;
    arAIN_46 : TItemAIN;
    arAIN_47 : TItemAIN;
    arAIN_48 : TItemAIN;
    arAIN_49 : TItemAIN;
    arAIN_50 : TItemAIN;
    arAIN_51 : TItemAIN;
    arAIN_52 : TItemAIN;
    arAIN_53 : TItemAIN;
    arAIN_54 : TItemAIN;
    arAIN_55 : TItemAIN;
    arAIN_56 : TItemAIN;
    arAIN_57 : TItemAIN;
    arAIN_58 : TItemAIN;
    arAIN_59 : TItemAIN;
    arAIN_60 : TItemAIN;
    arAIN_61 : TItemAIN;
    arAIN_62 : TItemAIN;
    arAIN_63 : TItemAIN;
    arERR_28 : TItemDIN;
    arERR_29 : TItemDIN;
    arERR_30 : TItemDIN;
    arERR_31 : TItemDIN;
    arERR_32 : TItemDIN;
    arERR_33 : TItemDIN;
    arERR_34 : TItemDIN;
    arERR_35 : TItemDIN;
    arERR_36 : TItemDIN;
    arERR_37 : TItemDIN;
    arERR_38 : TItemDIN;
    arERR_39 : TItemDIN;
    arERR_40 : TItemDIN;
    arERR_41 : TItemDIN;
    arERR_42 : TItemDIN;
    arERR_43 : TItemDIN;
    arERR_44 : TItemDIN;
    A2_14_err_mode : UINT;
    A2_15_err_mode : UINT;
    A3_10_err_mode : UINT;
    A3_11_err_mode : UINT;
    A3_12_err_mode : UINT;
    A3_13_err_mode : UINT;
    A3_14_err_mode : UINT;
    A3_15_err_mode : UINT;
    A3_1_err_mode : UINT;
    A3_2_err_mode : UINT;
    A3_3_err_mode : UINT;
    A3_4_err_mode : UINT;
    A3_5_err_mode : UINT;
    A3_6_err_mode : UINT;
    A3_7_err_mode : UINT;
    A3_8_err_mode : UINT;
    A3_9_err_mode : UINT;
    AI_0_dblValue : LREAL;
    AI_10_dblValue : LREAL;
    AI_11_dblValue : LREAL;
    AI_12_dblValue : LREAL;
    AI_13_dblValue : LREAL;
    AI_14_dblValue : LREAL;
    AI_15_dblValue : LREAL;
    AI_16_dblValue : LREAL;
    AI_17_dblValue : LREAL;
    AI_18_dblValue : LREAL;
    AI_19_dblValue : LREAL;
    AI_1_dblValue : LREAL;
    AI_20_dblValue : LREAL;
    AI_21_dblValue : LREAL;
    AI_22_dblValue : LREAL;
    AI_23_dblValue : LREAL;
    AI_24_dblValue : LREAL;
    AI_25_dblValue : LREAL;
    AI_26_dblValue : LREAL;
    AI_27_dblValue : LREAL;
    AI_28_dblValue : LREAL;
    AI_29_dblValue : LREAL;
    AI_2_dblValue : LREAL;
    AI_30_dblValue : LREAL;
    AI_31_dblValue : LREAL;
    AI_32_dblValue : LREAL;
    AI_33_dblValue : LREAL;
    AI_34_dblValue : LREAL;
    AI_35_dblValue : LREAL;
    AI_36_dblValue : LREAL;
    AI_37_dblValue : LREAL;
    AI_38_dblValue : LREAL;
    AI_39_dblValue : LREAL;
    AI_3_dblValue : LREAL;
    AI_40_dblValue : LREAL;
    AI_41_dblValue : LREAL;
    AI_42_dblValue : LREAL;
    AI_43_dblValue : LREAL;
    AI_44_dblValue : LREAL;
    AI_45_dblValue : LREAL;
    AI_46_dblValue : LREAL;
    AI_47_dblValue : LREAL;
    AI_48_dblValue : LREAL;
    AI_49_dblValue : LREAL;
    AI_4_dblValue : LREAL;
    AI_50_dblValue : LREAL;
    AI_51_dblValue : LREAL;
    AI_52_dblValue : LREAL;
    AI_53_dblValue : LREAL;
    AI_54_dblValue : LREAL;
    AI_55_dblValue : LREAL;
    AI_56_dblValue : LREAL;
    AI_57_dblValue : LREAL;
    AI_58_dblValue : LREAL;
    AI_59_dblValue : LREAL;
    AI_5_dblValue : LREAL;
    AI_60_dblValue : LREAL;
    AI_61_dblValue : LREAL;
    AI_62_dblValue : LREAL;
    AI_63_dblValue : LREAL;
    AI_64_dblValue : LREAL;
    AI_65_dblValue : LREAL;
    AI_66_dblValue : LREAL;
    AI_67_dblValue : LREAL;
    AI_6_dblValue : LREAL;
    AI_7_dblValue : LREAL;
    AI_8_dblValue : LREAL;
    AI_9_dblValue : LREAL;
    BS_Core1 : REAL;
    BS_Core2 : REAL;
    BS_Core3 : REAL;
    BS_Core4 : REAL;
    BS_FreeMemory : REAL;
    BS_Temp1 : REAL;
    BS_Temp2 : REAL;
    arAIN_64 : TItemAIN;
    arAIN_65 : TItemAIN;
    arAIN_66 : TItemAIN;
    arAIN_67 : TItemAIN;
  END_VAR

  (* Циклический опрос. Входные аналоговые параметры *)

  (********************************************* Модуль A2-14 ******************************************************)
  (* [A2-14, AI0-0] T_medi_statora_faza_1 *)
  fb_T_medi_statora_faza_1(arAIN := arAIN_0, strAI := ai.TStalisStatoraKanal1, err_mod:=arERR_28);
  AI_0_dblValue := arAIN_0.dblValue;

  (* [A2-14, AI0-1] T_medi_statora_faza_2 *)
  fb_T_medi_statora_faza_2(arAIN := arAIN_1, strAI := ai.TStalisStatoraKanal2, err_mod:=arERR_28);
  AI_1_dblValue := arAIN_1.dblValue;

  (* [A2-14, AI0-2] T_medi_statora_faza_3 *)
  fb_T_medi_statora_faza_3(arAIN := arAIN_2, strAI := ai.TStalisStatoraKanal3, err_mod:=arERR_28);
  AI_2_dblValue := arAIN_2.dblValue;

  (* [A2-14, AI0-3] T_stali_statora_faza_1 *)
  fb_T_stali_statora_faza_1(arAIN := arAIN_3, strAI := ai.TMediStatoraKanal1, err_mod:=arERR_28);
  AI_3_dblValue := arAIN_3.dblValue;

  A2_14_err_mode := arERR_28.wValue;

  (********************************************* Модуль A2-15 ******************************************************)

  (* [A2-15, AI1-0] T_stali_statora_faza_2 *)
  fb_T_stali_statora_faza_2(arAIN := arAIN_4, strAI := ai.TMediStatoraKanal2, err_mod:=arERR_29);
  AI_4_dblValue := arAIN_3.dblValue;

  (* [A2-15, AI1-1] T_stali_statora_faza_3 *)
  fb_T_stali_statora_faza_3(arAIN := arAIN_5, strAI := ai.TMediStatoraKanal3, err_mod:=arERR_29);
  AI_5_dblValue := arAIN_3.dblValue;

  (* [A2-15, AI1-2] T_goryachego_vozdyha_ed_t1 *)
  fb_T_goryachego_vozdyha_ed_t1(arAIN := arAIN_6, strAI := ai.TOpornogoPodshipnikaEDT_1, err_mod:=arERR_29);
  AI_6_dblValue := arAIN_3.dblValue;

  (* [A2-15, AI1-3]  T_goryachego_vozdyha_ed_t2 *)
  fb_T_goryachego_vozdyha_ed_t2(arAIN := arAIN_7, strAI := ai.TOpornoYpornogoPodshipnikaEDT_2, err_mod:=arERR_29);
  AI_7_dblValue := arAIN_3.dblValue;

  A2_15_err_mode := arERR_29.wValue;

  (********************************************* Модуль A3-1 ******************************************************)

  (* [A3-1, AI2-0]  T_holodnogo_vozdyha_ed_t1 *)
  fb_T_holodnogo_vozdyha_ed_t1(arAIN := arAIN_8, strAI := ai.TOpornoYpornogoPodshipnikaKolesaRedEDT_3, err_mod:=arERR_30);
  AI_8_dblValue := arAIN_3.dblValue;

  (* [A3-1, AI2-1] T_holodnogo_vozdyha_ed_t2 *)
  fb_T_holodnogo_vozdyha_ed_t2(arAIN := arAIN_9, strAI := ai.TOpornoYpornogoPodshipnikaKolesaRedHT_4, err_mod:=arERR_30);
  AI_9_dblValue := arAIN_3.dblValue;

  (* [A3-1, AI2-2] T_opornogo_podshipnika_electro_dvigatelia_t1 *)
  fb_T_OP_ED_t1(arAIN := arAIN_10, strAI := ai.TOpornogoPodshipnikaShesterniReduktoraT_5, err_mod:=arERR_30);
  AI_10_dblValue := arAIN_3.dblValue;

  (* [A3-1, AI2-3]  T_oporno_ypornogo_podshipnika_electro_dvigatelia_so_storony_redyctora_t2 *)
  fb_T_OYP_ED_so_storony_redyctora_t2(arAIN := arAIN_11, strAI := ai.TOpornogoPodshipnikaReduktoraHT_6, err_mod:=arERR_30);
  AI_11_dblValue := arAIN_3.dblValue;

  A3_1_err_mode := arERR_30.wValue;

  (********************************************* Модуль A3-2 ******************************************************)

  (* [A3-2, AI3-0]  T_oporno_ypornogo_podshipnika_kolesa_redyctora_so_storony_electro_dvigatelya_t3 *)
  fb_T_OYP_kolesa_ED_t3(arAIN := arAIN_12, strAI := ai.TOpornoYpornogoPodshipnikaNagnetateljaT_7_1, err_mod:=arERR_31);
  AI_12_dblValue := arAIN_3.dblValue;

  (* [A3-2, AI3-1]  T_opornogo_podshipnika_kolesa_redyctora_so_storony_nagnetatelya_t4 *)
  fb_T_OP_kolesa_nagnetatelya_t4(arAIN := arAIN_13, strAI := ai.TOpornoYpornogoPodshipnikaNagnetateljaT_7_2, err_mod:=arERR_31);
  AI_13_dblValue := arAIN_3.dblValue;

  (* [A3-2, AI3-2]  T_opornogo_podshipnika_shesterni_redyctora_so_storony_electro_dvigatelya_t5 *)
  fb_T_OP_shesterni_ED_t5(arAIN := arAIN_14, strAI := ai.TOpornoYpornogoPodshipnikaSvobodnogoKoncaNT_8_1, err_mod:=arERR_31);
  AI_14_dblValue := arAIN_3.dblValue;

  (* [A3-2, AI32-3]  T_opornogo_podshipnika_redyctora_so_storony_nagnetatelya_t6 *)
  fb_T_OP_redyctora_so_storony_nagnetatelya_t6(arAIN := arAIN_15, strAI := ai.TOpornoYpornogoPodshipnikaSvobodnogoKoncaNT_8_2, err_mod:=arERR_31);
  AI_15_dblValue := arAIN_3.dblValue;

  A3_2_err_mode := arERR_31.wValue;

  (********************************************* Модуль A3-3 ******************************************************)

  (* [A3-3, AI4-0]  T_oporno_ypornogo_podshipnika_nagnetatelya_so_storony_redyctora_t7_osnovnoi *)
  fb_T_OYP_nagnetatelya_so_storony_redyctora_t7_1(arAIN := arAIN_16, strAI := ai.TYpornogoPodshipnikaRavKolodokHT_9_1, err_mod:=arERR_32);
  AI_16_dblValue := arAIN_3.dblValue;

  (* [A3-3, AI4-1]  T_oporno_ypornogo_podshipnika_nagnetatelya_so_storony_redyctora_t7_rezervniy *)
  fb_T_OYP_nagnetatelya_so_storony_redyctora_t7_2(arAIN := arAIN_17, strAI := ai.TYpornogoPodshipnikaRavKolodokHT_9_2, err_mod:=arERR_32);
  AI_17_dblValue := arAIN_3.dblValue;

  (* [A3-3, AI4-2]  T_oporno_ypornogo_podshipnika_svobodnogo_konca_nagnetatelya_t8_osnovnoi *)
  fb_T_OYP_svobodnogo_konca_nagnetatelya_t8_1(arAIN := arAIN_18, strAI := ai.TYpornogoPodshipnikaNerabKolodokHT_10_1, err_mod:=arERR_32);
  AI_18_dblValue := arAIN_3.dblValue;

  (* [A3-3, AI4-3] T_oporno_ypornogo_podshipnika_svobodnogo_konca_nagnetatelya_t8_rezervniy *)
  fb_T_OYP_svobodnogo_konca_nagnetatelya_t8_2(arAIN := arAIN_19, strAI := ai.TYpornogoPodshipnikaNerabKolodokHT_10_2, err_mod:=arERR_32);
  AI_19_dblValue := arAIN_3.dblValue;

  A3_3_err_mode := arERR_32.wValue;

  (********************************************* Модуль A3-4 ******************************************************)

  (* [A3-4, AI5-0] T_ypornogo_podshipnika_rabochih_kolodok_nagnetatelya_t9 *)
  fb_T_YP_rabochih_kolodok_nagnetatelya_t9(arAIN := arAIN_20, strAI := ai.THolodnogoVozduhaEDKanall, err_mod:=arERR_33);
  AI_20_dblValue := arAIN_3.dblValue;

  (* [A3-4, AI5-1] T_ne_rabochih_kolodok_ypornogo_podshipnika_nagnetatelya_t10Т газа на входе нагнетателя *)
  fb_T_ne_rabochih_kolodok_YP_nagnetatelya_t10(arAIN := arAIN_21, strAI := ai.THolodnogoVozduhaEDKanal2, err_mod:=arERR_33);
  AI_21_dblValue := arAIN_3.dblValue;

  (* [A3-4, AI5-2]  T_gaz_in_nagnetatelia *)
  fb_T_gaz_in_nagnetatelia(arAIN := arAIN_22, strAI := ai.TGorjachegoVozduhaEDKanall, err_mod:=arERR_33);
  AI_22_dblValue := arAIN_3.dblValue;

  (* [A3-4, AI5-3] T_gaz_out_nagnetatelia *)
  fb_T_gaz_out_nagnetatelia(arAIN := arAIN_23, strAI := ai.TGorjachegoVozduhaEDKanal2, err_mod:=arERR_33);
  AI_23_dblValue := arAIN_3.dblValue;

  A3_3_err_mode := arERR_33.wValue;

  (********************************************* Модуль A3-5 ******************************************************)

  (* [A3-5, AI6-0] T_masla_do_ABO *)
  fb_T_masla_do_ABO(arAIN := arAIN_24, strAI := ai.TNArujnogoVozduha, err_mod:=arERR_34);
  AI_24_dblValue := arAIN_3.dblValue;

  (* [A3-5, AI6-1]  T_masla_posle_ABO *)
  fb_T_masla_posle_ABO(arAIN := arAIN_25, strAI := ai.TgazaNaVhodeH, err_mod:=arERR_34);
  AI_25_dblValue := arAIN_3.dblValue;

  (* [A3-5, AI6-2] T_masla_v_maslobake *)
  fb_T_masla_v_maslobake(arAIN := arAIN_26, strAI := ai.TgazaNaVyhodeH, err_mod:=arERR_34);
  AI_26_dblValue := arAIN_3.dblValue;

  AI_27_dblValue := arAIN_3.dblValue;

  A3_5_err_mode := arERR_34.wValue;

  (********************************************* Модуль A3-6 ******************************************************)

  (* [A1-8, AI7-0] T_masla_v_maslobake_nad_ten *)
  fb_T_masla_v_maslobake_nad_ten(arAIN := arAIN_28, strAI := ai.T_masla_v_maslobake_nad_ten, err_mod:=arERR_35);
  AI_28_dblValue := arAIN_3.dblValue;

  (* [A1-8, AI7-1] T_naryjnogo_vozdyxa_rezervniy *)
  fb_T_naryjnogo_vozdyxa(arAIN := arAIN_29, strAI := ai.T_naryjnogo_vozdyxa, err_mod:=arERR_35);
  AI_29_dblValue := arAIN_3.dblValue;

  (* [A1-8, AI7-2] T_vozduha_V_shkaf *)
  fb_T_vozduha_V_shkaf(arAIN := arAIN_30, strAI := ai.T_vozduha_V_shkaf, err_mod:=arERR_35);
  AI_30_dblValue := arAIN_30.dblValue;

  AI_31_dblValue := arAIN_31.dblValue;

  A3_6_err_mode := arERR_35.wValue;

  (********************************************* Модуль A3-7 ******************************************************)

  (* Резерв *)
  AI_32_dblValue := arAIN_32.dblValue;

  AI_33_dblValue := arAIN_33.dblValue;

  AI_34_dblValue := arAIN_34.dblValue;

  AI_35_dblValue := arAIN_35.dblValue;

  A3_7_err_mode := arERR_36.wValue;
  (********************************************* Модуль A3-8 ******************************************************)

  (* [A3-8, AI9-0]  Davlenie_impylsnogo_gaza *)
  fb_Davlenie_impylsnogo_gaza(arAIN := arAIN_36, strAI := ai.Davlenie_impylsnogo_gaza, err_mod:=arERR_37);
  AI_36_dblValue := arAIN_36.dblValue;

  (* [A3-8, AI9-1]  Yroven_masla_v_maslobake *)
  fb_Yroven_masla_v_maslobake(arAIN := arAIN_37, strAI := ai.Yroven_masla_v_maslobake, err_mod:=arERR_37);
  AI_37_dblValue := arAIN_37.dblValue;

  (* [A3-8, AI9-2]  Osevoi_sdvig_nagnetatelya_vpravo *)
  fb_Osevoi_sdvig_nagnetatelya_vpravo(arAIN := arAIN_38, strAI := ai.Osevoi_sdvig_nagnetatelya_vpravo, err_mod:=arERR_37);
  AI_38_dblValue := arAIN_38.dblValue;

  (* [A3-8, AI9-3]  Osevoi_sdvig_nagnetatelya_vlevo *)
  fb_Osevoi_sdvig_nagnetatelya_vlevo(arAIN := arAIN_39, strAI := ai.Osevoi_sdvig_nagnetatelya_vlevo, err_mod:=arERR_37);
  AI_39_dblValue := arAIN_39.dblValue;

  A3_8_err_mode := arERR_37.wValue;

  (********************************************* Модуль A3-9 ******************************************************)

  (* [A3-9, AI10-0]  Tok_statora *)
  fb_Tok_statora(arAIN := arAIN_40, strAI := ai.Tok_statora, err_mod:=arERR_38);
  AI_40_dblValue := arAIN_40.dblValue;

  (* [A3-9, AI10-1]  Kontrol_220_perem *)
  fb_Kontrol_220_perem(arAIN := arAIN_41, strAI := ai.Kontrol_220_perem, err_mod:=arERR_38);
  AI_41_dblValue := arAIN_41.dblValue;

  (* [A3-9, AI10-2]  Kontrol_220_post *)
  fb_Kontrol_220_post(arAIN := arAIN_42, strAI := ai.Kontrol_220_post, err_mod:=arERR_38);
  AI_42_dblValue := arAIN_42.dblValue;

  AI_43_dblValue := arAIN_43.dblValue;

  A3_9_err_mode := arERR_38.wValue;

  (********************************************* Модуль A3-10 ******************************************************)

  (* [A3-10, AI11-0] Davlenie_gaza_na_vhode_nagnetatelya *)
  fb_Davlenie_gaza_na_vhode_nagnetatelya(arAIN := arAIN_44, strAI := ai.Davlenie_gaza_na_vhode_nagnetatelya, err_mod:=arERR_39);
  AI_44_dblValue := arAIN_44.dblValue;

  (* [A3-10, AI11-1] Активная мощность *)
  fb_Davlenie_gaza_na_vihode_nagnetatelya(arAIN := arAIN_45, strAI := ai.Davlenie_gaza_na_vihode_nagnetatelya, err_mod:=arERR_39);
  AI_45_dblValue := arAIN_45.dblValue;

  (* [A3-10, AI11-2] Perepad_davleniya_maslo_gaz *)
  fb_Perepad_davleniya_maslo_gaz(arAIN := arAIN_46, strAI := ai.Perepad_davleniya_maslo_gaz, err_mod:=arERR_39);
  AI_46_dblValue := arAIN_46.dblValue;

  (* [A3-10, AI11-3] Davlenie_masla_posle_nasosa_yplotneniya *)
  fb_Davlenie_masla_posle_nasosa_yplotneniya(arAIN := arAIN_47, strAI := ai.Davlenie_masla_posle_nasosa_yplotneniya, err_mod:=arERR_39);
  AI_47_dblValue := arAIN_47.dblValue;

  A3_10_err_mode := arERR_39.wValue;

  (********************************************* Модуль A3-11 ******************************************************)

  (* [A3-11, AI12-0] Davlenie_masla_smazki_nizkoe *)
  fb_Davlenie_masla_smazki_nizkoe(arAIN := arAIN_48, strAI := ai.Davlenie_masla_smazki_nizkoe, err_mod:=arERR_40);
  AI_48_dblValue := arAIN_48.dblValue;

  (* [A3-11, AI12-1] Davlenie_masla_smazki_visokoe *)
  fb_Davlenie_masla_smazki_visokoe(arAIN := arAIN_49, strAI := ai.Davlenie_masla_smazki_visokoe, err_mod:=arERR_40);
  AI_49_dblValue := arAIN_49.dblValue;

  (* [A3-11, AI12-2] Davlenie_masla_smazki_posle_GNS *)
  fb_Davlenie_masla_smazki_posle_GNS(arAIN := arAIN_50, strAI := ai.Davlenie_masla_smazki_posle_GNS, err_mod:=arERR_40);
  AI_50_dblValue := arAIN_50.dblValue;

  (* [A3-11, AI12-3] Perepad_davleniya_gaza_na_konfyzore *)
  fb_Perepad_davleniya_gaza_na_konfyzore(arAIN := arAIN_51, strAI := ai.Perepad_davleniya_gaza_na_konfyzore, err_mod:=arERR_40);
  AI_51_dblValue := arAIN_51.dblValue;

  A3_11_err_mode := arERR_40.wValue;

  (********************************************* Модуль A3-12 ******************************************************)

  (* [A3-12, AI13-0] Perepad_davleniya_masla_na_maslyanom_filtre *)
  fb_Perepad_davleniya_masla_na_maslyanom_filtre(arAIN := arAIN_52, strAI := ai.Perepad_davleniya_masla_na_maslyanom_filtre, err_mod:=arERR_41);
  AI_52_dblValue := arAIN_52.dblValue;

  AI_53_dblValue := arAIN_53.dblValue;

  AI_54_dblValue := arAIN_54.dblValue;

  AI_55_dblValue := arAIN_55.dblValue;

  A3_12_err_mode := arERR_41.wValue;

  (********************************************* Модуль A3-13 ******************************************************)

  (* [A3-13, AI14-0] Vibroploskost_opornogo_podshipnika_electro_dvigatelya_t1 *)
  fb_Vibroskorost_OP_ED_t1(arAIN := arAIN_56, strAI := ai.Vibroskorost_OP_ED_t1, err_mod:=arERR_42);
  AI_56_dblValue := arAIN_56.dblValue;

  (* [A3-13, AI14-1] Vibroploskost_oporno_ypornogo_podshipnika_electro_dvigatelya_so_storony_redyctora_t2 *)
  fb_Vibroskorost_OYP_ED_so_storony_redyctora_t2(arAIN := arAIN_57, strAI := ai.Vibroskorost_OYP_ED_so_storony_redyctora_t2, err_mod:=arERR_42);
  AI_57_dblValue := arAIN_57.dblValue;

  (* [A3-13, AI14-2] Vibroploskost_oporno_ypornogo_podshipnika_kolesa_redyktora_so_storony_electro_dvigatelya_t3 *)
  fb_Vibroskorost_OYP_kolesa_ED_t3(arAIN := arAIN_58, strAI := ai.Vibroskorost_OYP_kolesa_ED_t3, err_mod:=arERR_42);
  AI_58_dblValue := arAIN_58.dblValue;

  (* [A3-13, AI14-3] Vibroploskost_oporno_ypornogo_podshipnika_kolesa_redyktora_so_storony_nagnetatelya_t4_rezerv *)
  fb_Vibroskorost_OP_kolesa_nagnetatelya_t4(arAIN := arAIN_59, strAI := ai.Vibroskorost_OP_kolesa_nagnetatelya_t4, err_mod:=arERR_42);
  AI_59_dblValue := arAIN_59.dblValue;

  A3_13_err_mode := arERR_42.wValue;

  (********************************************* Модуль A3-14 ******************************************************)

  (* [A3-14, AI14-0] Vibroploskost_opornogo_podshipnika_shesterni_redyktora_so_storony_nagnetatelya_t5_rezerv *)
  fb_Vibroskorost_OP_shesterni_ED_t5(arAIN := arAIN_60, strAI := ai.Vibroskorost_OP_shesterni_ED_t5, err_mod:=arERR_43);
  AI_60_dblValue := arAIN_60.dblValue;

  (* [A3-14, AI14-1] Vibroploskost_opornogo_podshipnika_shesterni_redyktora_so_storony_nagnetatelya_t6 *)
  fb_Vibroskorost_OP_shesterni_nagnetatelya_t6(arAIN := arAIN_61, strAI := ai.Vibroskorost_OP_shesterni_nagnetatelya_t6, err_mod:=arERR_43);
  AI_61_dblValue := arAIN_61.dblValue;

  AI_62_dblValue := arAIN_62.dblValue;

  AI_63_dblValue := arAIN_63.dblValue;

  A3_14_err_mode := arERR_43.wValue;

  (********************************************* Модуль A3-15 ******************************************************)

  (* Резерв *)
  AI_64_dblValue := arAIN_64.dblValue;

  AI_65_dblValue := arAIN_65.dblValue;

  AI_66_dblValue := arAIN_66.dblValue;

  AI_67_dblValue := arAIN_67.dblValue;

  A3_15_err_mode := arERR_44.wValue;

  (********************************************* Параметры с БС ******************************************************)
  (*
  BS_FreeMemory := LREAL_TO_REAL(arAIN_8.dblValue);
  BS_Temp1 := LREAL_TO_REAL(arAIN_9.dblValue);
  BS_Temp2 := LREAL_TO_REAL(arAIN_10.dblValue);
  BS_Core1 := LREAL_TO_REAL(arAIN_11.dblValue);
  BS_Core2 := LREAL_TO_REAL(arAIN_12.dblValue);
  BS_Core3 := LREAL_TO_REAL(arAIN_13.dblValue);
  BS_Core4 := LREAL_TO_REAL(arAIN_14.dblValue); *)
END_FUNCTION_BLOCK

FUNCTION_BLOCK proc_AI_Init
  VAR_INPUT
    init : BOOL;
  END_VAR
  VAR
    stAI_Ini : fb_AI_Init;
    inits : UINT;
  END_VAR
  VAR_INPUT
    initiales : UINT;
  END_VAR
  VAR_EXTERNAL
    ai : AiConfig;
  END_VAR

  (* Инициализация начало. Входные аналоговые параметры *)

  inits := 0; (* Флаг необходимости инициализации структур-дескрипторов *)

  (********************************************* Модуль A2-14 ******************************************************)
  (* [A2-14, AI0-0] T_medi_statora_faza_1 *)
  stAI_Ini(data_Ini := TRUE, dLL := 0.0, dHL := 150.0,
  ISVALIDREF_HW := TRUE, dHW := 130.0, aperturFilter:= 0.5,
  strAI := ai.TStalisStatoraKanal1);
  inits := inits + BOOL_TO_UINT(stAI_Ini.Init);
